// SIMATIC STEP 7 (V5.x) project Line1A_Nozzle_20101204
// CPU: CPU 315-2 DP
// station: Hardware
// station: SIMATIC 300(1)
// station: P_ADR_BUS
// station: P_ADR_BUS
// station: Configuration
// program: S7 Program(6)
// program: Controllo camera doppio
// program: Backup_prima_della_mod
// program: SIMODRIVE 611U

SYMBOL_TABLE
"Z10"	C 10	COUNTER	// Counter
"Z11"	C 11	COUNTER	// Counter
"Z12"	C 12	COUNTER	// Counter
"Z13"	C 13	COUNTER	// Counter
"DI_Balluff1"	DB 5	FB 20	// DB Instance of FB20
"DatiOP170B"	DB 7	DB 7	// PLC<->OP170B interface
"Timer"	DB 20	DB 20
"DBWork"	DB 21	DB 21
"coordinate"	DB 22	DB 22
"DB180"	DB 180	FB 24	// DB instance FB24 AsseY
"DB181"	DB 181	FB 24	// DB instance FB24 AsseX
"DBWork2"	DB 200	DB 200
"Asse_611U"	FB 16	FB 16	// Axis 611U management
"BALLUFF"	FB 20	FB 20	// BALLUFF Reader/Writer management
"FB24 - Gestione Mov Assi"	FB 24	FB 24	// GESTIONE ASSI STAZIONE
"NormalizzazioneAnalogico"	FC 7	FC 7	// Normalization of a analog value
"FC11 - STATUS"	FC 11	FC 11	// Sensors and proximity state
"FC12 - GENERAL"	FC 12	FC 12	// General management
"FC13 - MANUAL"	FC 13	FC 13	// Manual commands
"FC14 - AUTOMATIC"	FC 14	FC 14	// Automatic cycle management
"FC16 - ALARMS"	FC 16	FC 16	// Alarms management
"FC17 - OPERATOR PANNEL"	FC 17	FC 17	// Operator pannel management
"FC18 - OUTPUTS"	FC 18	FC 18	// Outputs management
"FC19 - REPOSITIONING"	FC 19	FC 19	// Repositioning management
"FC - AUTOMATIC"	FC 24	FC 24
"FC50 - TEACH-IN"	FC 50	FC 50
"FC51 - TYPE TOOL"	FC 51	FC 51
"FC52 - SYSTEM VISION"	FC 52	FC 52
"FC53 - REWORK"	FC 53	FC 53
"FC81 - GEST AXIS"	FC 81	FC 81	// Management axis
"FC117 - ERROR TOOL"	FC 117	FC 117
"TimeOut"	FC 800	FC 800	// Management TimeOut movimenti
"E0.0"	I 0.0	BOOL	// THERMAL SWTCH_ASPIRATOR_MTR
"E0.1"	I 0.1	BOOL	// 230 Vac power supply circuit braker
"E0.2"	I 0.2	BOOL	// 230 VAC PS CKT BRAKER
"E0.3"	I 0.3	BOOL	// Welding Machine OK
"E0.4"	I 0.4	BOOL	// Reserve
"E0.5"	I 0.5	BOOL	// AUXILIXARY ON
"DOOR CLOSE"	I 0.6	BOOL	// Reserve
"E0.7"	I 0.7	BOOL	// SAFETY BARRIER
"E1.0"	I 1.0	BOOL	// CYCLE_START
"E1.1"	I 1.1	BOOL	// AUTO_MANUAL
"E1.2"	I 1.2	BOOL	// COMPRESSED AIR
"E1.3"	I 1.3	BOOL	// AXIS RESET_POS
"E1.4"	I 1.4	BOOL	// Rotary table motor thermal switch
"E1.5"	I 1.5	BOOL	// LCK_UNLCK_DOORS_PB
"E1.6"	I 1.6	BOOL	// Reserve
"E1.7"	I 1.7	BOOL	// DRIVE TEMP
"E2.0"	I 2.0	BOOL	// STOP_CYCLE_PB
"E2.1"	I 2.1	BOOL	// Doors Closed & Locked
"E2.2"	I 2.2	BOOL	// Safety Barrier OK
"E2.3"	I 2.3	BOOL	// WELDING_TORCH_DWN
"E2.4"	I 2.4	BOOL	// WELDING_TORCH_UP
"E2.5"	I 2.5	BOOL	// ROTARY_TABLE_ZERO
"E2.6"	I 2.6	BOOL	// ROTARY_TABLE_ZERO1
"E2.7"	I 2.7	BOOL	// Reserve
"E3.0"	I 3.0	BOOL	// VEN DETECTOR_FWD
"E3.1"	I 3.1	BOOL	// VEN DETECTOR_REV
"E3.2"	I 3.2	BOOL	// VEN DETECTOR_DWN
"E3.3"	I 3.3	BOOL	// VEN DETECTOR_UP
"E3.4"	I 3.4	BOOL	// ROTARY_TABLE_CAM
"E3.5"	I 3.5	BOOL	// Reserve
"E3.6"	I 3.6	BOOL	// Reserve
"E3.7"	I 3.7	BOOL	// Reserve
"e5.0"	I 5.0	BOOL	// Lever Detector System - bit 0
"e5.1"	I 5.1	BOOL	// Lever Detector System - bit 1
"e5.2"	I 5.2	BOOL	// Lever Detector System - bit 2
"e5.3"	I 5.3	BOOL	// Lever Detector System - bit 3
"e5.4"	I 5.4	BOOL	// Lever Detector System - bit 4
"e5.5"	I 5.5	BOOL	// Lever Detector System - bit 5
"e5.6"	I 5.6	BOOL	// Lever Detector System - bit 6
"e5.7"	I 5.7	BOOL	// Lever Detector System - bit 7
"e6.0"	I 6.0	BOOL	// Lever Detector System - bit 8
"e6.1"	I 6.1	BOOL	// Lever Detector System - bit 9
"e6.2"	I 6.2	BOOL	// Lever Detector System - bit 10
"e6.3"	I 6.3	BOOL	// Lever Detector System - bit 11 - 12è13
"e6.4"	I 6.4	BOOL	// Lever Detector System - bit 12
"e6.5"	I 6.5	BOOL	// Lever Detector System - bit 13
"e6.6"	I 6.6	BOOL	// Lever Detector System - bit 14
"e6.7"	I 6.7	BOOL	// Lever Detector System - Vane Assy Total Number
"EXSTRACTOR_HIGH"	I 7.2	BOOL
"EXSTRACTOR_LOW"	I 7.3	BOOL
"TABLE_LCK_CYCLINDER_UP"	I 7.4	BOOL
"TABLE_LCK_CYCLINDER_DWN"	I 7.5	BOOL
"E32.0"	I 32.0	BOOL	// Push-button start cycle (on load position)
"E32.1"	I 32.1	BOOL	// Push button stop cycle
"E32.2"	I 32.2	BOOL	// Aut/Man Selector
"E32.3"	I 32.3	BOOL	// Reserve
"E32.4"	I 32.4	BOOL	// Reserve
"E32.5"	I 32.5	BOOL	// Lock/Unlock doors Push Button
"E32.6"	I 32.6	BOOL	// Reserve
"E32.7"	I 32.7	BOOL	// Air Presence
"E34.0"	I 34.0	BOOL	// Cam Table
"E34.1"	I 34.1	BOOL	// Reserve
"E34.2"	I 34.2	BOOL	// Reserve
"E34.3"	I 34.3	BOOL	// Reserve
"E34.4"	I 34.4	BOOL	// Table locker cylinder  up
"E34.5"	I 34.5	BOOL	// Table locker cylinder down
"E34.6"	I 34.6	BOOL	// Exstractor High
"E34.7"	I 34.7	BOOL	// Extractor Low
"E35.0"	I 35.0	BOOL	// Torch Welding low
"E35.1"	I 35.1	BOOL	// Torch Welding high
"E35.2"	I 35.2	BOOL	// Home Assy
"E35.3"	I 35.3	BOOL	// 1 --> PP1 on welding ; 0 --> PP2 on welding
"E35.4"	I 35.4	BOOL	// Detect components Control group High
"E35.5"	I 35.5	BOOL	// Detect components Control group Low
"E35.6"	I 35.6	BOOL	// Detect components Control group forward
"E35.7"	I 35.7	BOOL	// Detect components Control group backward
"E36.0"	I 36.0	BOOL	// Reserve not mounted
"E36.1"	I 36.1	BOOL	// Reserve not mounted
"E36.2"	I 36.2	BOOL	// Reserve not mounted
"E36.3"	I 36.3	BOOL	// Reserve not mounted
"E36.4"	I 36.4	BOOL	// Reserve not mounted
"E36.5"	I 36.5	BOOL	// Reserve not mounted
"E36.6"	I 36.6	BOOL	// Reserve not mounted
"E36.7"	I 36.7	BOOL	// Reserve not mounted
"E52.0"	I 52.0	BOOL	// Lever Detector System - bit 0
"E52.1"	I 52.1	BOOL	// Lever Detector System - bit 1
"E52.2"	I 52.2	BOOL	// Lever Detector System - bit 2
"E52.3"	I 52.3	BOOL	// Lever Detector System - bit 3
"E52.4"	I 52.4	BOOL	// Lever Detector System - bit 4
"E52.5"	I 52.5	BOOL	// Lever Detector System - bit 5
"E52.6"	I 52.6	BOOL	// Lever Detector System - bit 6
"E52.7"	I 52.7	BOOL	// Lever Detector System - bit 7
"E53.0"	I 53.0	BOOL	// Lever Detector System - bit 8
"E53.1"	I 53.1	BOOL	// Lever Detector System - bit 9
"E53.2"	I 53.2	BOOL	// Lever Detector System - bit 10
"E53.3"	I 53.3	BOOL	// Lever Detector System - bit 11 - 12è13
"E53.4"	I 53.4	BOOL	// Lever Detector System - bit 12
"E53.5"	I 53.5	BOOL	// Lever Detector System - bit 13
"E53.6"	I 53.6	BOOL	// Lever Detector System - bit 14
"E53.7"	I 53.7	BOOL	// Lever Detector System - Vane Assy Total Number
"E64.0"	I 64.0	BOOL	// VOSION SYSTEM OK
"E64.1"	I 64.1	BOOL	// Busy
"E64.2"	I 64.2	BOOL	// Or
"E64.3"	I 64.3	BOOL	// Error
"E64.4"	I 64.4	BOOL	// Gate
"E64.5"	I 64.5	BOOL	// Strobe trigger 0 out
"E64.6"	I 64.6	BOOL	// Strobe trigger 1 out
"E64.7"	I 64.7	BOOL	// DO0
"E65.0"	I 65.0	BOOL	// DO1
"E65.1"	I 65.1	BOOL	// DO2
"E65.2"	I 65.2	BOOL	// DO3
"E65.3"	I 65.3	BOOL	// DO4
"E65.4"	I 65.4	BOOL	// DO5
"E65.5"	I 65.5	BOOL	// DO6
"E65.6"	I 65.6	BOOL	// DO7
"E65.7"	I 65.7	BOOL	// DO8
"M0.0"	M 0.0	BOOL	// Clock 0,1 s
"M0.1"	M 0.1	BOOL	// Clock 0,2 s
"M0.2"	M 0.2	BOOL	// Clock 0,4 s
"M0.3"	M 0.3	BOOL	// Clock 0,5 s
"M0.4"	M 0.4	BOOL	// Clock 0,8 s
"M0.5"	M 0.5	BOOL	// Clock 1 s
"M0.6"	M 0.6	BOOL	// Clock 1,6 s
"M0.7"	M 0.7	BOOL	// Clock 2 s
"Off"	M 1.0	BOOL	// Merker always OFF
"On"	M 1.1	BOOL	// Merker always ON
"ToDo"	M 1.2	BOOL
"Bypass"	M 1.3	BOOL	// Merker that indicates a bypass forced of the code
"BypassPC"	M 1.4	BOOL	// Merker for bypass control handshake with PC supervision
"Clock_P"	M 1.5	BOOL	// Positiv pulse of clock
"Clock_N"	M 1.6	BOOL	// Negativ pulse of code
"Clock_10s"	M 1.7	BOOL	// 10 seconds clock
"M2.0"	M 2.0	BOOL	// Occhio
"BPSupervisor"	M 3.0	BOOL	// By Pass del supervisore
"Auxiliary_ON"	M 10.0	BOOL	// Auxiliary ON
"COMPRESSED_AIR"	M 10.1	BOOL	// Compressed Air
"SHIELDS_OK"	M 10.2	BOOL	// Schermi Chiusi e bloccati
"MACHINE_ON"	M 10.3	BOOL	// Machine OK
"START_POS"	M 11.0	BOOL	// Machine in initial positon
"START_POS_MEM"	M 11.1	BOOL	// mem initial position
"M11.2"	M 11.2	BOOL	// Manual Mode Selected
"SEMI"	M 11.3	BOOL	// Selezione modo semi automatico
"AUT"	M 11.4	BOOL	// Automatic Mode Selected
"START"	M 12.0	BOOL	// Start machine
"START_PULSE"	M 12.1	BOOL	// Pulse of start push-button
"SINGLE_CYCLE"	M 12.2	BOOL	// 1=ciclo singolo 0=ciclo continuo
"ALARM"	M 12.3	BOOL	// Alarm
"END_CYCLE"	M 12.4	BOOL	// Automatic cycle finished
"CmdMan_Av"	M 12.5	BOOL	// Forward manual command
"CmdMan_Ind"	M 12.6	BOOL	// Backward manual command
"STOP_BUTTON"	M 12.7	BOOL	// STATUS - stop button
"M13.0"	M 13.0	BOOL	// STATUS - Lock/Unlock doors Push Button
"M14.0"	M 14.0	BOOL	// Mem Lever Detector System - bit 0
"M14.1"	M 14.1	BOOL	// Mem Lever Detector System - bit 1
"M14.2"	M 14.2	BOOL	// Mem Lever Detector System - bit 2
"M14.3"	M 14.3	BOOL	// Mem Lever Detector System - bit 3
"M14.4"	M 14.4	BOOL	// Mem Lever Detector System - bit 4
"M14.5"	M 14.5	BOOL	// Mem Lever Detector System - bit 5
"M14.6"	M 14.6	BOOL	// Mem Lever Detector System - bit 6
"M14.7"	M 14.7	BOOL	// Mem Lever Detector System - bit 7
"M15.0"	M 15.0	BOOL	// Mem Lever Detector System - bit 8
"M15.1"	M 15.1	BOOL	// Mem Lever Detector System - bit 9
"M15.2"	M 15.2	BOOL	// Mem Lever Detector System - bit 10
"M15.3"	M 15.3	BOOL	// Mem Lever Detector System - bit 11
"M15.4"	M 15.4	BOOL	// Mem Lever Detector System - bit 12
"M15.5"	M 15.5	BOOL	// Mem Lever Detector System - bit 13
"M15.6"	M 15.6	BOOL	// Mem Lever Detector System - bit 14 (Roller)
"M15.7"	M 15.7	BOOL	// Mem Lever Detector System - bit 15
"M16.0"	M 16.0	BOOL	// mem Reworked Parts
"M16.1"	M 16.1	BOOL	// Disable Extractor if Rework
"M16.2"	M 16.2	BOOL	// Part on table 1 welding
"M16.3"	M 16.3	BOOL	// Part on Table 2 Welding
"M16.4"	M 16.4	BOOL	// Table can ROTATE
"M16.5"	M 16.5	BOOL	// Extractor can MOVE
"M16.6"	M 16.6	BOOL	// OK Extract
"M16.7"	M 16.7	BOOL	// Manual PAge Active
"M17.2"	M 17.2	BOOL	// Rework
"M17.3"	M 17.3	BOOL	// Vane no welding
"M17.4"	M 17.4	BOOL	// PP2 - OUT
"M17.5"	M 17.5	BOOL	// PP1 - OUT
"M17.6"	M 17.6	BOOL	// AUX - F R E E
"M17.7"	M 17.7	BOOL	// AUX - F R E E
"M18.0"	M 18.0	BOOL	// AUX - F R E E
"M18.1"	M 18.1	BOOL	// AUX - F R E E
"M18.2"	M 18.2	BOOL	// AUX - F R E E
"M18.3"	M 18.3	BOOL	// AUX - F R E E
"M18.4"	M 18.4	BOOL	// AUX - F R E E
"M18.5"	M 18.5	BOOL	// AUX - F R E E
"M18.6"	M 18.6	BOOL	// AUX - F R E E
"M18.7"	M 18.7	BOOL	// AUX - F R E E
"M19.0"	M 19.0	BOOL	// AUX - F R E E
"M19.1"	M 19.1	BOOL	// AUX - F R E E
"M19.2"	M 19.2	BOOL	// AUX - F R E E
"M19.3"	M 19.3	BOOL	// AUX - F R E E
"M19.4"	M 19.4	BOOL	// AUX - F R E E
"M19.5"	M 19.5	BOOL	// AUX - F R E E
"M19.6"	M 19.6	BOOL	// AUX - F R E E
"M19.7"	M 19.7	BOOL	// AUX - F R E E
"M20.0"	M 20.0	BOOL	// AUX - F R E E
"M20.1"	M 20.1	BOOL	// AUX - F R E E
"M20.2"	M 20.2	BOOL	// Presence of tool to assembly nozzle
"M20.3"	M 20.3	BOOL	// AUX - F R E E
"M20.4"	M 20.4	BOOL	// Tension OK
"M20.5"	M 20.5	BOOL	// AUX - F R E E
"M20.6"	M 20.6	BOOL	// AUX - F R E E
"M20.7"	M 20.7	BOOL	// AUX-Man
"M21.0"	M 21.0	BOOL	// STATUS - Mem Component pinched on Workrest - FC1
"Mem E34.5"	M 21.1	BOOL	// Mem Component pinched on Workrest - FC2
"M21.2"	M 21.2	BOOL	// AUX - F R E E
"M21.3"	M 21.3	BOOL	// AUX - F R E E
"M21.4"	M 21.4	BOOL	// Aux Alarm
"Warning"	M 21.5	BOOL	// Warning
"ResetAlarm"	M 21.6	BOOL	// Reset alarm
"Repos"	M 21.7	BOOL	// Repositioning
"M22.0"	M 22.0	BOOL	// STATUS - Table locker up
"M22.1"	M 22.1	BOOL	// STATUS - Table locker Down
"CmdMan_Av_Pulse"	M 22.2	BOOL	// Pulse of forward manual command
"CmdMan_Ind_Pulse"	M 22.3	BOOL	// Pulse of backward manual command
"M22.4"	M 22.4	BOOL	// Forward command
"M22.5"	M 22.5	BOOL	// Backward command
"CmdMan_Esg"	M 22.6	BOOL	// Memory of manual command executed
"CicloInCorso"	M 22.7	BOOL	// Automatic cycle in course
"M23.0"	M 23.0	BOOL	// Mem Start
"StopAEndCycle"	M 23.1	BOOL
"ChangeFunc"	M 23.2	BOOL	// Pulse change operation mode
"PresencePz"	M 23.3	BOOL
"SafetyBarrier_KO"	M 23.5	BOOL	// STATUS - Security bar KO
"M24.0"	M 24.0	BOOL	// STATUS - Torch Welding low
"M24.1"	M 24.1	BOOL	// STATUS - Torch Welding high
"M24.2"	M 24.2	BOOL	// STATUS -
"M24.3"	M 24.3	BOOL	// STATUS -
"M24.4"	M 24.4	BOOL	// STATUS - Cam table
"M24.5"	M 24.5	BOOL	// 1 --> PP1 on welding ;0 --> PP2 on welding
"M25.0"	M 25.0	BOOL	// Position Rotation 0°
"M25.1"	M 25.1	BOOL	// Position Rotation 180°
"M25.2"	M 25.2	BOOL	// Pos 0° e camma OK
"M25.3"	M 25.3	BOOL	// Pos 180° e camma OK
"M25.7"	M 25.7	BOOL	// Pulse Cam
"M26.1"	M 26.1	BOOL	// Table is FREE
"M26.2"	M 26.2	BOOL	// STATUS - System Detector Up
"M26.3"	M 26.3	BOOL	// STATUS - System Detector Lower
"M26.4"	M 26.4	BOOL	// STATUS - Detector work position
"M26.5"	M 26.5	BOOL	// STATUS - Detector park position
"M26.6"	M 26.6	BOOL	// STATUS - Exstractor High
"M26.7"	M 26.7	BOOL	// STATUS - Extractor low
"M28.0"	M 28.0	BOOL	// STATUS - DO1SYSTEM VISION
"M28.1"	M 28.1	BOOL	// STATUS - DO2 SYSTEM VISION
"M28.2"	M 28.2	BOOL	// STATUS - DO3 SYSTEM VISION
"M28.3"	M 28.3	BOOL	// STATUS - DO4 SYSTEM VISION
"M29.0"	M 29.0	BOOL	// STATUS - Run System Vision
"M29.1"	M 29.1	BOOL	// STATUS - Busy System Vision
"M29.2"	M 29.2	BOOL	// STATUS - OK System Vision
"M29.3"	M 29.3	BOOL	// STATUS - Error System Vision
"M29.4"	M 29.4	BOOL	// STATUS - Gate System Vision
"M29.6"	M 29.6	BOOL	// STATUS - DO1 SYSTEM VISION
"M29.7"	M 29.7	BOOL	// STATUS - DO0 SYSTEM VISION
"M30.0"	M 30.0	BOOL	// MAN - Table Rotation Forward
"M30.1"	M 30.1	BOOL	// MAN - Table Rotation Backward
"M30.2"	M 30.2	BOOL	// MAN - Jog + AsseY
"M30.3"	M 30.3	BOOL	// MAN - Jog - AsseY
"M30.4"	M 30.4	BOOL	// MAN - Jog + AsseX
"M30.5"	M 30.5	BOOL	// MAN - Jog - AsseX
"M30.6"	M 30.6	BOOL	// MAN - Forward SD
"M30.7"	M 30.7	BOOL	// MAN - Backward SD
"M31.0"	M 31.0	BOOL	// MAN - High SD
"M31.1"	M 31.1	BOOL	// MAN - Low SD
"M31.2"	M 31.2	BOOL	// MAN - High TW
"M31.3"	M 31.3	BOOL	// MAN - Low TW
"M31.4"	M 31.4	BOOL	// MAN - Extractor High
"M31.5"	M 31.5	BOOL	// MAN - Extractor down
"M31.6"	M 31.6	BOOL	// MAN - ON\OFF TW
"M31.7"	M 31.7	BOOL	// MAN - START/STOP WM
"M32.0"	M 32.0	BOOL	// Man  -  Start Torch W"elding
"M32.1"	M 32.1	BOOL	// MAN - Test Arco Gas Ok
"M32.2"	M 32.2	BOOL	// MAN - Test Arco Gas
"M32.3"	M 32.3	BOOL	// MAN - Torch Welding Temp Ok
"M32.4"	M 32.4	BOOL	// MAN - low table locker cylinder
"M32.5"	M 32.5	BOOL	// MAN - up table locker cylinder
"M32.6"	M 32.6	BOOL	// MAN - Welding
"M32.7"	M 32.7	BOOL	// MAN - Free
"M33.0"	M 33.0	BOOL	// MAN - Free
"M33.1"	M 33.1	BOOL	// MAN - Free
"M33.2"	M 33.2	BOOL	// MAN - Free
"M33.3"	M 33.3	BOOL	// MAN - Free
"M33.4"	M 33.4	BOOL	// MAN - Free
"M33.5"	M 33.5	BOOL	// MAN - Free
"M33.6"	M 33.6	BOOL	// MAN - Free
"M33.7"	M 33.7	BOOL	// MAN - Free
"M34.0"	M 34.0	BOOL	// MAN - Memory for rotation table
"M34.1"	M 34.1	BOOL	// MAN - Memory back rotation table
"M34.2"	M 34.2	BOOL	// MAN - Free
"M34.3"	M 34.3	BOOL	// MAN - Free
"M34.4"	M 34.4	BOOL	// MAN - Free
"M34.5"	M 34.5	BOOL	// MAN - Free
"M34.6"	M 34.6	BOOL	// MAN - Free
"M34.7"	M 34.7	BOOL	// MAN - Free
"M40.0"	M 40.0	BOOL	// RIP - Start repositioning
"M40.1"	M 40.1	BOOL	// RIP - Start reposit CamTable
"M40.2"	M 40.2	BOOL	// RIP - Cam Table
"M40.3"	M 40.3	BOOL	// RIP - System Detector vertical
"M40.4"	M 40.4	BOOL	// RIP - System Detector horizontal
"M40.5"	M 40.5	BOOL	// RIP - torch welding
"M40.6"	M 40.6	BOOL	// RIP - estractor
"M40.7"	M 40.7	BOOL	// RIP - Axis X and Y
"M41.0"	M 41.0	BOOL	// RIP - low table locker cylinder
"M41.1"	M 41.1	BOOL	// RIP - up table locker cylinder
"M41.2"	M 41.2	BOOL	// RIP - Free
"M41.3"	M 41.3	BOOL	// RIP - Free
"M41.4"	M 41.4	BOOL	// RIP - Free
"M41.5"	M 41.5	BOOL	// RIP - Free
"M41.6"	M 41.6	BOOL	// RIP - Free
"M41.7"	M 41.7	BOOL	// RIP - Free
"M42.0"	M 42.0	BOOL	// RIP - Free
"M42.1"	M 42.1	BOOL	// RIP - Table locker
"M42.2"	M 42.2	BOOL	// RIP - Free
"M42.3"	M 42.3	BOOL	// RIP - Free
"M42.4"	M 42.4	BOOL	// RIP - Free
"M42.5"	M 42.5	BOOL	// RIP - Free
"M42.6"	M 42.6	BOOL	// RIP - Free
"M42.7"	M 42.7	BOOL	// RIP - Free
"M50.0"	M 50.0	BOOL	// AUT - Table forward Side A
"M50.1"	M 50.1	BOOL	// AUT - Table backward Side B
"M50.2"	M 50.2	BOOL	// AUT - System Detector Forward
"M50.3"	M 50.3	BOOL	// AUT - System Detector Backward
"M50.4"	M 50.4	BOOL	// AUT - System Detector Low
"M50.5"	M 50.5	BOOL	// AUT - System Detector High
"M50.6"	M 50.6	BOOL	// AUT - welding down
"M50.7"	M 50.7	BOOL	// AUT - welding up
"M51.0"	M 51.0	BOOL	// AUT - Free
"M51.1"	M 51.1	BOOL	// AUT - Free
"M51.2"	M 51.2	BOOL	// AUT - Free
"M51.3"	M 51.3	BOOL	// AUT - Estractor High
"M51.4"	M 51.4	BOOL	// AUT - Estractor Low
"M51.5"	M 51.5	BOOL	// AUT - Free
"M51.6"	M 51.6	BOOL	// AUT - Free
"M51.7"	M 51.7	BOOL	// AUT - Free
"M52.0"	M 52.0	BOOL	// AUT -Temp  welding OK
"M52.1"	M 52.1	BOOL	// AUT - welding now
"M52.2"	M 52.2	BOOL	// AUT - Trigger System Vision
"M52.3"	M 52.3	BOOL	// AUT - ligth up
"M52.4"	M 52.4	BOOL	// AUT - Test Arc
"M52.5"	M 52.5	BOOL	// AUT - Test Arc Gas Ok
"M52.6"	M 52.6	BOOL	// AUT - low table locker cylinder
"M52.7"	M 52.7	BOOL	// AUT - up table locker cylinder
"M53.0"	M 53.0	BOOL	// AUT - Table locker Up
"M53.1"	M 53.1	BOOL	// AUT - Table locker Down
"M60.0"	M 60.0	BOOL	// STEP - 1:Table Forward
"M60.1"	M 60.1	BOOL	// STEP - 2:System Detector Forward
"M60.2"	M 60.2	BOOL	// STEP 3- System Detector Low
"M60.3"	M 60.3	BOOL	// STEP - 3 Check Nozzle Component
"M60.4"	M 60.4	BOOL	// STEP - 5 System detector High
"M60.5"	M 60.5	BOOL	// STEP 6 - System Detector Bacward
"M60.6"	M 60.6	BOOL	// STEP -7 welding down on point
"M60.7"	M 60.7	BOOL	// STEP - welding OK
"M61.0"	M 61.0	BOOL	// STEP - All welding is effectuated
"M61.1"	M 61.1	BOOL	// STEP - Photo Executed
"M61.2"	M 61.2	BOOL	// STEP - Axis in position 0
"M61.3"	M 61.3	BOOL	// STEP - point for welding receive
"M61.4"	M 61.4	BOOL	// STEP - welding up after work
"M61.5"	M 61.5	BOOL	// STEP - Welding in progress
"M61.6"	M 61.6	BOOL	// STEP - Start Rotation Table
"M61.7"	M 61.7	BOOL	// STEP - Photo without error
"M62.0"	M 62.0	BOOL	// STEP - Mem Reset Table
"M62.1"	M 62.1	BOOL	// STEP - Free
"M62.2"	M 62.2	BOOL	// STEP - Table cylinder up
"M62.3"	M 62.3	BOOL	// STEP - Free
"M62.4"	M 62.4	BOOL	// STEP - Free
"M62.5"	M 62.5	BOOL	// STEP - Free
"M62.6"	M 62.6	BOOL	// STEP - Free
"M62.7"	M 62.7	BOOL	// STEP - Photo Executed
"M63.0"	M 63.0	BOOL	// STEP - Nozzle Extracted
"M63.1"	M 63.1	BOOL	// STEP - Table Cylinder Low
"M63.6"	M 63.6	BOOL	// STEP - receive point photo
"M66.0"	M 66.0	BOOL	// STEP - photo 1 is NO good
"M66.1"	M 66.1	BOOL	// STEP - photo 2 is NO good
"M66.4"	M 66.4	BOOL	// STEP - Axis in position
"M66.6"	M 66.6	BOOL	// STEP - Execute 2th photo
"M66.7"	M 66.7	BOOL	// STEP - All photo is NO Good
"M67.0"	M 67.0	BOOL	// STEP - Axis Y in position
"M67.1"	M 67.1	BOOL	// STEP - Axis X in position
"M70.0"	M 70.0	BOOL	// Nozzle components Ok
"M70.1"	M 70.1	BOOL	// memNozzle-components Ok
"M70.2"	M 70.2	BOOL	// Component of Nozzle KO
"M70.3"	M 70.3	BOOL	// error assembling su PP1
"M70.4"	M 70.4	BOOL	// error assembling su PP2
"M71.0"	M 71.0	BOOL	// System Detector in Pos initial
"M72.0"	M 72.0	BOOL	// ready for welding
"M73.0"	M 73.0	BOOL	// Enable velocity for repositioning
"M74.0"	M 74.0	BOOL	// Output SV enable
"M74.1"	M 74.1	BOOL	// piece good
"M74.2"	M 74.2	BOOL	// piece reject
"M75.0"	M 75.0	BOOL	// Enable movement axis for teach in
"M75.1"	M 75.1	BOOL	// TeachIn OK
"M76.0"	M 76.0	BOOL	// position welding receive
"MEM Welding Machine OK"	M 80.0	BOOL
"Type_PP1_10_vane"	M 90.0	BOOL	// PP1-10 presence
"Type_PP2_9_vane"	M 90.1	BOOL	// presence PP2 -11 welding
"Type_PP3_9_vane"	M 90.2	BOOL	// presence PP3 - 9welding
"Type_PP4_13_vane"	M 90.3	BOOL	// presence PP4 - 13 Welding
"AUT STEP 1"	M 160.0	BOOL
"AUT STEP 2"	M 160.1	BOOL
"AUT STEP 3"	M 160.2	BOOL
"AUT STEP 4"	M 160.3	BOOL
"AUT STEP 5"	M 160.4	BOOL
"AUT STEP 6"	M 160.5	BOOL
"AUT STEP 7"	M 160.6	BOOL
"AUT STEP 8"	M 160.7	BOOL
"AUT STEP 9"	M 161.0	BOOL
"AUT STEP10"	M 161.1	BOOL
"AUT STEP11"	M 161.2	BOOL
"AUT STEP12"	M 161.3	BOOL
"AUT STEP13"	M 161.4	BOOL
"AUT STEP14"	M 161.5	BOOL
"AUT STEP15"	M 161.6	BOOL
"AUT STEP16"	M 161.7	BOOL
"AUT STEP17"	M 162.0	BOOL
"AUT STEP18"	M 162.1	BOOL
"AUT STEP19"	M 162.2	BOOL
"AUT STEP20"	M 162.3	BOOL
"AUT STEP21"	M 162.4	BOOL
"AUT STEP22"	M 162.5	BOOL
"AUT STEP23"	M 162.6	BOOL
"AUT STEP24"	M 162.7	BOOL
"AUT STEP25"	M 163.0	BOOL
"AUT STEP26"	M 163.1	BOOL
"AUT STEP27"	M 163.2	BOOL
"AUT STEP28"	M 163.3	BOOL
"AUT STEP29"	M 163.4	BOOL
"AUT STEP30"	M 163.5	BOOL
"Clock 0.5 S"	M 200.3	BOOL
"Clock 1s"	M 200.5	BOOL
"M254.0"	M 254.0	BOOL	// Front Command HOME
"M254.1"	M 254.1	BOOL	// Front Command END
"M256.0"	M 256.0	BOOL	// Pulse
"M256.2"	M 256.2	BOOL	// Pulse
"M256.6"	M 256.6	BOOL	// Pulse
"M256.7"	M 256.7	BOOL	// Pulse
"M340.0"	M 340.0	BOOL	// AXIS Y:STOP MOVE
"M340.1"	M 340.1	BOOL	// AXIS Y:START POSITIONING
"M340.2"	M 340.2	BOOL	// AXIS Y:START SEARCH HOME
"M340.3"	M 340.3	BOOL	// AXIS Y:START POSITIONING ON HOME
"M340.4"	M 340.4	BOOL	// AXIS X:COMMAND JOG PLUS
"M340.5"	M 340.5	BOOL	// AXIS X:COMANDO JOG LESS
"M341.0"	M 341.0	BOOL	// AXIS Y:ACHIEVED LOCATION
"M341.1"	M 341.1	BOOL	// AXIS Y:REFERED AXIS
"M341.2"	M 341.2	BOOL	// AXIS Y:AXIS LOCATION ON HOME
"M341.3"	M 341.3	BOOL	// AXIS Y:AXIS STOP NONE COMMAND PROGRESS
"M341.4"	M 341.4	BOOL	// AXIS Y:SETTING SETTING IN MOTION OK
"M341.5"	M 341.5	BOOL	// AXIS Y:ALLRM SETTING IN MOTION
"M342.0"	M 342.0	BOOL	// AXIS Y:AXIS ON CAM OF  REFERENCE
"M342.1"	M 342.1	BOOL	// AXIS Y:AXIS ON OVER RACE NEGATIVE HARDWARE
"M342.2"	M 342.2	BOOL	// AXIS Y:AXIS ON OVER RACE POSITIVE HARDWARE
"M342.3"	M 342.3	BOOL	// AXIS Y:COMMAND BRAKE PARKING
"M342.4"	M 342.4	BOOL	// AXIS Y:AXIS ON OVER RACE NEGATIVE SOFTWARE
"M342.5"	M 342.5	BOOL	// AXIS Y:AXIS ON OVER RACE POSITIVE SOFTWARE
"M342.6"	M 342.6	BOOL	// AXIS Y:POSSIBLE MOVE AXIS
"M342.7"	M 342.7	BOOL	// AXIS Y:INITIAL LOCATION AXIS
"M343.0"	M 343.0	BOOL	// AXIS Y:START POSITIONING INCREMENTAL
"M346.0"	M 346.0	BOOL	// AXIS X:STOP MOVE
"M346.1"	M 346.1	BOOL	// AXIS X:START POSITIONING
"M346.2"	M 346.2	BOOL	// AXIS X:START SEARCH HOME
"M346.3"	M 346.3	BOOL	// AXIS X:START POSITIONING ON HOME
"M346.4"	M 346.4	BOOL	// AXIS Y:COMMAND JOG PLUS
"M346.5"	M 346.5	BOOL	// AXIS Y:COMANDO JOG LESS
"M347.0"	M 347.0	BOOL	// AXIS X:ACHIEVED LOCATION
"M347.1"	M 347.1	BOOL	// AXIS X:REFERED AXIS
"M347.2"	M 347.2	BOOL	// AXIS X:AXIS LOCATION ON HOME
"M347.3"	M 347.3	BOOL	// AXIS X:AXIS STOP NONE COMMAND PROGRESS
"M347.4"	M 347.4	BOOL	// AXIS X:SETTING SETTING IN MOTION OK
"M347.5"	M 347.5	BOOL	// AXIS X:ALLRM SETTING IN MOTION
"M348.0"	M 348.0	BOOL	// AXIS X:AXIS ON CAM OF  REFERENCE
"M348.1"	M 348.1	BOOL	// AXIS X:AXIS ON OVER RACE NEGATIVE HARDWARE
"M348.2"	M 348.2	BOOL	// AXIS X:AXIS ON OVER RACE POSITIVE HARDWARE
"M348.3"	M 348.3	BOOL	// AXIS X:COMMAND BRAKE PARKING
"M348.4"	M 348.4	BOOL	// AXIS X:AXIS ON OVER RACE NEGATIVE SOFTWARE
"M348.5"	M 348.5	BOOL	// AXIS X:AXIS ON OVER RACE POSITIVE SOFTWARE
"M348.6"	M 348.6	BOOL	// AXIS X:POSSIBLE MOVE AXIS
"M348.7"	M 348.7	BOOL	// AXIS X:INITIAL LOCATION AXIS
"M349.0"	M 349.0	BOOL	// AXIS X:START POSITIONING INCREMENTAL
"Photo 2 executed"	M 500.0	BOOL	// m61.1
"TriggerVisSystem2"	M 500.1	BOOL
"ErroreCamera"	M 500.7	BOOL
"M1000.0"	M 1000.0	BOOL	// AUX
"M1000.1"	M 1000.1	BOOL	// AUX
"M1000.2"	M 1000.2	BOOL	// AUX
"M1000.3"	M 1000.3	BOOL	// AUX
"M1000.4"	M 1000.4	BOOL	// AUX
"M1000.5"	M 1000.5	BOOL	// AUX
"M1000.6"	M 1000.6	BOOL	// AUX
"M1000.7"	M 1000.7	BOOL	// AUX
"M1001.0"	M 1001.0	BOOL	// AUX
"M1001.1"	M 1001.1	BOOL	// AUX
"M1001.2"	M 1001.2	BOOL	// AUX
"M1001.3"	M 1001.3	BOOL	// AUX
"M1001.4"	M 1001.4	BOOL	// AUX
"M1001.5"	M 1001.5	BOOL	// AUX
"M1001.6"	M 1001.6	BOOL	// AUX
"M1001.7"	M 1001.7	BOOL	// AUX
"M1002.0"	M 1002.0	BOOL	// AUX
"M1002.1"	M 1002.1	BOOL	// AUX
"M1002.2"	M 1002.2	BOOL	// AUX
"M1002.3"	M 1002.3	BOOL	// AUX
"M1002.4"	M 1002.4	BOOL	// AUX
"M1002.5"	M 1002.5	BOOL	// AUX
"M1002.6"	M 1002.6	BOOL	// AUX
"M1002.7"	M 1002.7	BOOL	// AUX
"M1003.0"	M 1003.0	BOOL	// AUX
"M1003.1"	M 1003.1	BOOL	// AUX
"M1003.2"	M 1003.2	BOOL	// AUX
"M1003.3"	M 1003.3	BOOL	// AUX
"M1003.4"	M 1003.4	BOOL	// AUX
"M1003.5"	M 1003.5	BOOL	// AUX
"M1003.6"	M 1003.6	BOOL	// AUX
"M1003.7"	M 1003.7	BOOL	// AUX
"M1004.0"	M 1004.0	BOOL	// AUX
"M1004.1"	M 1004.1	BOOL	// AUX
"M1004.2"	M 1004.2	BOOL	// AUX
"M1004.3"	M 1004.3	BOOL	// AUX
"M1004.4"	M 1004.4	BOOL	// AUX
"M1004.5"	M 1004.5	BOOL	// AUX
"M1004.6"	M 1004.6	BOOL	// AUX
"M1004.7"	M 1004.7	BOOL	// AUX
"M1005.0"	M 1005.0	BOOL	// AUX
"M1005.1"	M 1005.1	BOOL	// AUX
"M1005.2"	M 1005.2	BOOL	// AUX
"M1005.3"	M 1005.3	BOOL	// AUX
"M1005.4"	M 1005.4	BOOL	// AUX
"M1005.5"	M 1005.5	BOOL	// AUX
"M1005.6"	M 1005.6	BOOL	// AUX
"M1005.7"	M 1005.7	BOOL	// AUX
"M1006.0"	M 1006.0	BOOL	// AUX
"M1006.1"	M 1006.1	BOOL	// AUX
"M1006.2"	M 1006.2	BOOL	// AUX
"M1006.3"	M 1006.3	BOOL	// AUX
"M1006.4"	M 1006.4	BOOL	// AUX
"M1006.5"	M 1006.5	BOOL	// AUX
"M1006.6"	M 1006.6	BOOL	// AUX
"M1006.7"	M 1006.7	BOOL	// AUX
"M1007.0"	M 1007.0	BOOL	// AUX
"M1007.1"	M 1007.1	BOOL	// AUX
"M1007.2"	M 1007.2	BOOL	// AUX
"M1007.3"	M 1007.3	BOOL	// AUX
"M1007.4"	M 1007.4	BOOL	// AUX
"M1007.5"	M 1007.5	BOOL	// AUX
"M1007.6"	M 1007.6	BOOL	// AUX
"M1007.7"	M 1007.7	BOOL	// AUX
"M1008.0"	M 1008.0	BOOL	// AUX
"M1008.1"	M 1008.1	BOOL	// AUX
"M1008.2"	M 1008.2	BOOL	// AUX
"M1008.3"	M 1008.3	BOOL	// AUX
"M1008.4"	M 1008.4	BOOL	// AUX
"M1008.5"	M 1008.5	BOOL	// AUX
"M1008.6"	M 1008.6	BOOL	// AUX
"M1008.7"	M 1008.7	BOOL	// AUX
"M1009.0"	M 1009.0	BOOL	// AUX
"M1009.1"	M 1009.1	BOOL	// AUX
"M1009.2"	M 1009.2	BOOL	// AUX
"M1009.3"	M 1009.3	BOOL	// AUX
"M1009.4"	M 1009.4	BOOL	// AUX
"M1009.5"	M 1009.5	BOOL	// AUX
"M1009.6"	M 1009.6	BOOL	// AUX
"M1009.7"	M 1009.7	BOOL	// AUX
"FPAuxON_force_Axis_reset"	M 1900.0	BOOL
"Luce telecamera"	M 1900.2	BOOL
"AppoFP_M1900.3"	M 1900.3	BOOL
"Soffio Camera"	M 1900.4	BOOL
"Manual_cameralight_on"	M 1900.5	BOOL
"M2034.0"	M 2034.0	BOOL	// Key Start from pannell
"M2034.1"	M 2034.1	BOOL	// Key Finish from pannell
"M2034.2"	M 2034.2	BOOL	// Key Teach In from Pannell
"M2034.5"	M 2034.5	BOOL	// Key Enter teach from pannel
"M2034.6"	M 2034.6	BOOL	// Key Exit teach from pannel
"M2034.7"	M 2034.7	BOOL	// Key Rite from pannell
"M2035.0"	M 2035.0	BOOL	// Key Start from Teach In page
"M2035.1"	M 2035.1	BOOL	// Key Welding Run from pannel
"M2035.2"	M 2035.2	BOOL	// Key ACK on page 21 from pannell
"MB2046"	MB 2046	BYTE	// white byte
"MD30"	MD 30	DWORD	// DWORD Manual Commands
"MD100"	MD 100	DWORD	// temp
"MD588"	MD 588	DINT	// temporary for X point
"MD592"	MD 592	DINT	// temporary for X point
"MD596"	MD 596	DINT	// target X
"MD600"	MD 600	DINT	// target Y
"MD620"	MD 620	DWORD	// InsertPointX
"MD624"	MD 624	DWORD	// InsertPointY
"MD650"	MD 650	DINT	// axis X actual position
"MD654"	MD 654	DINT	// axis Y actual posiion
"SaldEffet"	MW 110	WORD	// number welding make
"MW120"	MW 120	INT	// number welding make
"MW300"	MW 300	INT	// number point to want go
"MW2042"	MW 2042	INT	// temp for clock
"MAIN PROGRAM"	OB 1	OB 1	// Main Program
"I/O_FLT1"	OB 82	OB 82	// I/O Point Fault 1
"RACK_FLT"	OB 86	OB 86	// Loss of Rack Fault
"COMPLETE RESTART"	OB 100	OB 100	// Complete Restart
"MOD_ERR"	OB 122	OB 122	// Module Access Error
"A0.0"	Q 0.0	BOOL	// Red Lamp
"A0.1"	Q 0.1	BOOL	// Yellow Lamp
"A0.2"	Q 0.2	BOOL	// Green Lamp
"A0.3"	Q 0.3	BOOL	// Lock doors relay
"A0.4"	Q 0.4	BOOL	// Simodrive Reset realy
"A0.5"	Q 0.5	BOOL	// Reserve
"A0.6"	Q 0.6	BOOL	// Reserve
"A0.7"	Q 0.7	BOOL	// Reserve
"A1.0"	Q 1.0	BOOL	// Enable Coral Vacuum
"A1.1"	Q 1.1	BOOL	// Test Gas Arco Pilota
"A1.2"	Q 1.2	BOOL	// Forward table rotation
"A1.3"	Q 1.3	BOOL	// Backward table rotation
"A1.4"	Q 1.4	BOOL	// Enable Axis X
"A1.5"	Q 1.5	BOOL	// Enable Axis Y
"A1.6"	Q 1.6	BOOL	// Start Welding
"A1.7"	Q 1.7	BOOL	// Ignition torch
"A2.0"	Q 2.0	BOOL	// Reserve
"A2.1"	Q 2.1	BOOL	// Reserve
"A2.2"	Q 2.2	BOOL	// Reserve
"A2.3"	Q 2.3	BOOL	// Reserve
"A2.4"	Q 2.4	BOOL	// Reserve
"A2.5"	Q 2.5	BOOL	// Reserve
"A2.6"	Q 2.6	BOOL	// Reserve
"A2.7"	Q 2.7	BOOL	// Reserve
"A3.0"	Q 3.0	BOOL	// Reserve
"A3.1"	Q 3.1	BOOL	// Reserve
"A3.2"	Q 3.2	BOOL	// Reserve
"A3.3"	Q 3.3	BOOL	// Reserve
"A3.4"	Q 3.4	BOOL	// Reserve
"A3.5"	Q 3.5	BOOL	// Reserve
"A3.6"	Q 3.6	BOOL	// Reserve
"A3.7"	Q 3.7	BOOL	// Reserve
"SIMODRIVE_RESET"	Q 12.0	BOOL
"BUZZER"	Q 12.1	BOOL
"Torch Welding Machin"	Q 12.2	BOOL	// Down
"Torch Welding MachinE"	Q 12.3	BOOL	// UP
"TABLE_LCKER_DWN"	Q 12.4	BOOL
"Table locker cylinder up"	Q 12.5	BOOL
"FWD_LEVER_DETECT_SYS"	Q 12.6	BOOL
"REV_LEVER_DETECT_SYS"	Q 12.7	BOOL
"UP_lever detector system"	Q 13.0	BOOL
"DW_lever detector sys"	Q 13.1	BOOL
"UP_Down _Extractor"	Q 13.2	BOOL
"_soffio_telecamera"	Q 13.3	BOOL
"DRIVE_ENABLE"	Q 13.5	BOOL
"ENABLE_Y_AXIS"	Q 13.6	BOOL
"ENABLE_X_AXIS"	Q 13.7	BOOL
"STOP_CYCLE_LAMP"	Q 14.3	BOOL
"START_CYCLE_LAMP"	Q 14.4	BOOL
"a14.5"	Q 14.5	BOOL
"ACCESES_BARRIER_LAMP"	Q 14.6	BOOL
"Enable Coral Vacuum"	Q 17.0	BOOL
"FWD_TABLE_ROTATION"	Q 17.1	BOOL
"REVERSE_TABLE_ROTATION"	Q 17.2	BOOL
"IGNITION_TORCH"	Q 17.5	BOOL
"START_WELDING"	Q 17.6	BOOL
"Test Gas Arc Pilota"	Q 17.7	BOOL
"PLC READY"	Q 18.0	BOOL	// ADDITION
"_Illumin_telecamera"	Q 18.1	BOOL
"PIECE_REFUSE"	Q 18.3	BOOL
"RED_LAMP"	Q 18.4	BOOL
"PIECE_GOOD"	Q 18.5	BOOL
"Lamp_Door_Locked"	Q 18.6	BOOL
"LOCK_DOORS_RELAY"	Q 18.7	BOOL
"A32.0"	Q 32.0	BOOL	// Lamp Start cycle
"A32.1"	Q 32.1	BOOL	// Lamp Stop cycle
"A32.2"	Q 32.2	BOOL	// Piece Good
"A32.3"	Q 32.3	BOOL	// Piece Refuse
"A32.4"	Q 32.4	BOOL	// Unlocked doors
"A32.5"	Q 32.5	BOOL	// Emergency Lamp
"A32.6"	Q 32.6	BOOL	// Access barrier Lamp
"A32.7"	Q 32.7	BOOL	// Buzzer
"A33.0"	Q 33.0	BOOL	// Reserve
"A33.1"	Q 33.1	BOOL	// Reserve
"A33.2"	Q 33.2	BOOL	// Reserve
"A33.3"	Q 33.3	BOOL	// Reserve
"A33.4"	Q 33.4	BOOL	// Reserve not mounted
"A33.5"	Q 33.5	BOOL	// Reserve not mounted
"A33.6"	Q 33.6	BOOL	// Reserve not mounted
"A33.7"	Q 33.7	BOOL	// Reserve not mounted
"A34.0"	Q 34.0	BOOL	// Forward lever detector System
"A34.1"	Q 34.1	BOOL	// Backward lever detector System
"A34.2"	Q 34.2	BOOL	// Down lever detector system
"A34.3"	Q 34.3	BOOL	// Up lever detector system
"A34.4"	Q 34.4	BOOL	// Down Torch Welding Machine
"A34.5"	Q 34.5	BOOL	// Up Torch Welding Machine
"A34.6"	Q 34.6	BOOL	// Down Extractor
"A34.7"	Q 34.7	BOOL	// Up Extractor
"A35.0"	Q 35.0	BOOL	// Table locker down
"A35.1"	Q 35.1	BOOL	// Table locker up
"A35.2"	Q 35.2	BOOL	// Reserve
"A35.3"	Q 35.3	BOOL	// Reserve
"A35.4"	Q 35.4	BOOL	// Reserve
"A35.5"	Q 35.5	BOOL	// Reserve
"A35.6"	Q 35.6	BOOL	// Reserve
"A35.7"	Q 35.7	BOOL	// Reserve
"A64.0"	Q 64.0	BOOL	// Reset
"A64.1"	Q 64.1	BOOL	// Trigger
"A64.2"	Q 64.2	BOOL	// Data Send Request
"A64.3"	Q 64.3	BOOL	// DI0
"A64.4"	Q 64.4	BOOL	// DI1
"A64.5"	Q 64.5	BOOL	// DI2
"A64.6"	Q 64.6	BOOL	// DI3
"A64.7"	Q 64.7	BOOL	// DI4
"A65.0"	Q 65.0	BOOL	// DI5
"A65.1"	Q 65.1	BOOL	// DI6
"A65.2"	Q 65.2	BOOL	// DI7
"A65.3"	Q 65.3	BOOL	// DI8
"A65.4"	Q 65.4	BOOL	// DI9
"A65.5"	Q 65.5	BOOL	// Reserve
"A65.6"	Q 65.6	BOOL	// Reserve
"A65.7"	Q 65.7	BOOL	// Reserve
"TON"	SFB 4	SFB 4	// Generate an On Delay
"READ_CLK"	SFC 1	SFC 1	// Read System Clock
"DPRD_DAT"	SFC 14	SFC 14	// Read Consistent Data of a Standard DP Slave
"DPWR_DAT"	SFC 15	SFC 15	// Write Consistent Data to a Standard DP Slave
"BLKMOV"	SFC 20	SFC 20	// Copy Variables
"FILL"	SFC 21	SFC 21	// Initialize a Memory Area
"CREAT_DB"	SFC 22	SFC 22	// Create Data Block
"DIS_AIRT"	SFC 41	SFC 41	// Delay the Higher Priority Interrupts and Asynchronous Errors
"EN_AIRT"	SFC 42	SFC 42	// Enable Higher Priority Interrupts and Asynchronous Errors
"STP"	SFC 46	SFC 46	// Change the CPU to STOP
"LGC_GADR"	SFC 49	SFC 49	// Query the Module Slot Belonging to a Logical Address
"RDSYSST"	SFC 51	SFC 51	// Read a System Status List or Partial List
"WR_REC"	SFC 58	SFC 58	// Write Data Record
"RD_REC"	SFC 59	SFC 59	// Read a Data Record
"T2"	T 2	TIMER
"T3"	T 3	TIMER	// Time for Component Start UP
"T10"	T 10	TIMER	// Delay
"T11"	T 11	TIMER
"T12"	T 12	TIMER	// delay next step
"T13"	T 13	TIMER	// Delay
"T14"	T 14	TIMER	// timer for delay KO
"T15"	T 15	TIMER	// Delay
"T16"	T 16	TIMER	// Delay
"T17"	T 17	TIMER	// timer delay
"T18"	T 18	TIMER	// Delay
"T19"	T 19	TIMER	// delay
"T20"	T 20	TIMER	// timer delay
"T21"	T 21	TIMER	// Time Test Arc
"T22"	T 22	TIMER	// Delay
"T23"	T 23	TIMER	// Timer for repositioning
"T24"	T 24	TIMER	// Delay make 2th photo
"T25"	T 25	TIMER	// delay
"T26"	T 26	TIMER	// time for reset output rotation table
"T27"	T 27	TIMER	// Timer for Executed Photo
"T28"	T 28	TIMER	// Delay for entry in teach in mode
"T29"	T 29	TIMER	// delay for reset both axis
"T30"	T 30	TIMER	// timer dealy
"T31"	T 31	TIMER	// MAN - time for welding
"T32"	T 32	TIMER	// MAN - time for welding UP
"T33"	T 33	TIMER	// Delay
"T34"	T 34	TIMER	// Time Test Arco
"T35"	T 35	TIMER	// Delay
"T36"	T 36	TIMER	// delay for cam not present
"T37"	T 37	TIMER	// Time Torch Welding Ok
"T38"	T 38	TIMER	// timer reset alarms axis X
"T39"	T 39	TIMER	// timer reset alarms axis Y
"T40"	T 40	TIMER	// Time Torch Welding Ok
"T41"	T 41	TIMER	// delay alarm air pressure
"T42"	T 42	TIMER	// Timer stop welding
"T43"	T 43	TIMER	// Timer welding Manual
"T44"	T 44	TIMER	// Delay
"T45"	T 45	TIMER	// timer for upgrade value
"T46"	T 46	TIMER	// delay enable axis Ytimer reset alarms axis X
"T47"	T 47	TIMER	// delay
"T48"	T 48	TIMER	// delay enable axis Ytimer reset alarms axis Y
"T50"	T 50	TIMER	// Delay
"T51"	T 51	TIMER
"T52"	T 52	TIMER	// wait after rotation table
"T53"	T 53	TIMER	// delay for chek camera point
"T54"	T 54	TIMER	// delay turn OFF Buzzer
"T60"	T 60	TIMER	// Delay for entry in teach in mode
"T61"	T 61	TIMER	// delay go in position for 2th photo
"T62"	T 62	TIMER	// delay for axis in position
"T63"	T 63	TIMER	// Delay
"T_SystemDetectorDW"	T 70	TIMER
"T_SystemDetector_UP"	T 71	TIMER
"T90"	T 90	TIMER	// delay allarm for Simodrive
"VAT_1"	VAT 1	
"Coordinate_saldatura"	VAT 2	
"I/O System Vision"	VAT 3	
"Saldatrice"	VAT 4	
"VAT_12"	VAT 5	
"VAT_PUNTI_AVV"	VAT 6	
"VAT_PUNTI_AVV_2"	VAT 7	
"DB22_SaldaturaSilv"	VAT 8	
"DB22_Sald_PP1"	VAT 9	
"VAT_tool check"	VAT 10	
"VAT_Balluff"	VAT 11	
"ASSE_P"	VAT 12	
"DB22_Sald_PP3"	VAT 13	
"VAT_Point"	VAT 14	
"VAT_Point 16"	VAT 15	
"DB22_Sald_PP16"	VAT 16	
"VAT_17"	VAT 17	
"Tipo portapezzo"	VAT 18	
"VAT_Daniele"	VAT 19	
END_SYMBOL_TABLE

FUNCTION_BLOCK "Asse_611U"	// FB 16
TITLE = Axis 611U management
VERSION : 0.1
VAR_INPUT
  IO_LAddr : INT ;	//Logic address of the inputs/outputs
END_VAR
VAR
  In_Profibus : STRUCT 	//Inputs from 611U (via Profibus)
   PKW : STRUCT 	//Parameter area of the Profibus telegram
    PKE : WORD ;
    IND : WORD ;
    PWE : DINT ;
   END_STRUCT ;
   PZD : STRUCT 	//Process data area of the Profibus telegram
    ZSW1 : STRUCT 	//Status word 1
     Bit8 : BOOL ;	//Following error (0=following error outside the window error)
     Bit9 : BOOL ;	//DP control requested (1=DP master is requested to accept control)
     Bit10 : BOOL ;	//Reference position reached (1=end of traversing block reached)
     Bit11 : BOOL ;	//Reference point set (1=axis is referenced)
     Bit12 : BOOL ;	//Setpoint acknowledge (1=the traversing task is processed)
     Bit13 : BOOL ;	//Drive stationery (1=drive is not in movement)
     Bit14 : BOOL ;	//External block change selected
     Bit15 : BOOL ;	//Request passive referencing
     Bit0 : BOOL ;	//Ready to switch-on (1=ready to power-up)
     Bit1 : BOOL ;	//Ready or no fault (1=drive ready or no fault present)
     Bit2 : BOOL ;	//Controller enable (1=speed controller active and setpoint can be accepted)
     Bit3 : BOOL ;	//Fault present (1=fault present)
     Bit4 : BOOL ;	//No OFF2 (1=OFF2 not present)
     Bit5 : BOOL ;	//No OFF3 (1=OFF3 not present)
     Bit6 : BOOL ;	//Switch-on inhibit (1=power-on inhibit)
     Bit7 : BOOL ;	//Alarm present (1=alarm present)
    END_STRUCT ;
    AktSatz : STRUCT 	//Actual block status word
     Bit8 : BOOL ;	//Reserved
     Bit9 : BOOL ;	//Reserved
     Bit10 : BOOL ;	//Reserved
     Bit11 : BOOL ;	//Reserved
     Bit12 : BOOL ;	//Reserved
     Bit13 : BOOL ;	//Reserved
     Bit14 : BOOL ;	//Reserved
     Bit15 : BOOL ;	//MDI Active
     Bit0 : BOOL ;	//Bit 0 block selected
     Bit1 : BOOL ;	//Bit 1 block selected
     Bit2 : BOOL ;	//Bit 2 block selected
     Bit3 : BOOL ;	//Bit 3 block selected
     Bit4 : BOOL ;	//Bit 4 block selected
     Bit5 : BOOL ;	//Bit 5 block selected
     Bit6 : BOOL ;	//Reserved
     Bit7 : BOOL ;	//Reserved
    END_STRUCT ;
    PosZsw : STRUCT 	//Position status word
     Bit8 : BOOL ;	//Cam switching signal 1
     Bit9 : BOOL ;	//Cam switching signal 2
     Bit10 : BOOL ;	//Direct output 1 via the traversing block
     Bit11 : BOOL ;	//Direct output 2 via the traversing block
     Bit12 : BOOL ;	//Fixed endstop reached
     Bit13 : BOOL ;	//Fixed endstop clamping torque reached
     Bit14 : BOOL ;	//Traverse to fixed endstop active
     Bit15 : BOOL ;	//Teach-In executed
     Bit0 : BOOL ;	//Tracking mode active (1=tracking mode active)
     Bit1 : BOOL ;	//Velocity limiting (1=velocity is limited)
     Bit2 : BOOL ;	//Setpoint stationary (1=axis stationary on the setpoint side)
     Bit3 : BOOL ;	//In synchronism (1=slave drive is synchronized with the master drive)
     Bit4 : BOOL ;	//Axis moves forwards
     Bit5 : BOOL ;	//Axis moves backwards
     Bit6 : BOOL ;	//Minus software limit switch actuated
     Bit7 : BOOL ;	//Plus software limit switch actuated
    END_STRUCT ;
    ZSW2 : STRUCT 	//Status word 2
     Bit8 : BOOL ;	//Suppress fault 608 active
     Bit9 : BOOL ;	//n.u. (used only in the n-set mode)
     Bit10 : BOOL ;	//n.u. (used only in the n-set mode)
     Bit11 : BOOL ;	//n.u. (used only in the n-set mode)
     Bit12 : BOOL ;	//Slave sign-of-life
     Bit13 : BOOL ;	//Slave sign-of-life
     Bit14 : BOOL ;	//Slave sign-of-life
     Bit15 : BOOL ;	//Slave sign-of-life
     Bit0 : BOOL ;	//Bit 0 parameter set
     Bit1 : BOOL ;	//Bit 1 parameter set
     Bit2 : BOOL ;	//Bit 2 parameter set
     Bit3 : BOOL ;	//First speed setpoint filter inactive
     Bit4 : BOOL ;	//Rump-function generator inactive
     Bit5 : BOOL ;	//Open holding brake
     Bit6 : BOOL ;	//Integrator inhibit
     Bit7 : BOOL ;	//Parking axis selected
    END_STRUCT ;
    XretrP : DINT ;	//Actual position value
    DIG_IN : STRUCT 	//Digital inputs status
     Bit8 : BOOL ;
     Bit9 : BOOL ;
     Bit10 : BOOL ;
     Bit11 : BOOL ;
     Bit12 : BOOL ;
     Bit13 : BOOL ;
     Bit14 : BOOL ;
     Bit15 : BOOL ;
     Bit0 : BOOL ;	//Axis on home cam
     Bit1 : BOOL ;	//Axis on minus extra-corse limit switch
     Bit2 : BOOL ;	//Axis on plus extra-corse limit switch
     Bit3 : BOOL ;
     Bit4 : BOOL ;
     Bit5 : BOOL ;
     Bit6 : BOOL ;
     Bit7 : BOOL ;
    END_STRUCT ;
   END_STRUCT ;
  END_STRUCT ;
  Out_Profibus : STRUCT 	//Outputs to 611U (via Profibus)
   PKW : STRUCT 	//Parameter area of the Profibus telegram
    PKE : WORD ;
    IND : WORD ;
    PWE : DINT ;
   END_STRUCT ;
   PZD : STRUCT 	//Process data area of the Profibus telegram
    STW1 : STRUCT 	//Control word 1
     Bit8 : BOOL ;	//JOG1 (1=the drive traverse with the speed in P0108)
     Bit9 : BOOL ;	//JOG2 (1=the drive traverse with the speed in P0109)
     Bit10 : BOOL ;	//Control requested (Should be set 1 when ZSW1.9=1)
     Bit11 : BOOL ;	//Stop referencing (1=start the referencing point approach)
     Bit12 : BOOL ;	//Opening the holding brake for test purposes
     Bit13 : BOOL ;	//External block change (With a edge the external block changing is initiated)
     Bit14 : BOOL ;	//Reserved
     Bit15 : BOOL ;	//Request passive referencing
     Bit0 : BOOL ;	//OFF1 (1=enable)
     Bit1 : BOOL ;	//OFF2 (1=enable)
     Bit2 : BOOL ;	//OFF3 (1=enable)
     Bit3 : BOOL ;	//Pulse inhibit (0=the motor stop for inertia)
     Bit4 : BOOL ;	//Reject travel task (0=stop the motor and delete the distance to go)
     Bit5 : BOOL ;	//Intermediate stop (0=stop the motor but the process is continued with 0/1 edge)
     Bit6 : BOOL ;	//Activate travel task (With a edge the traversing block selected is started)
     Bit7 : BOOL ;	//Reset the fault memory (1=Reset the fault memory)
    END_STRUCT ;
    SatzAnw : STRUCT 	//Block selection control word
     Bit8 : BOOL ;	//Reserved
     Bit9 : BOOL ;	//Reserved
     Bit10 : BOOL ;	//Reserved
     Bit11 : BOOL ;	//Reserved
     Bit12 : BOOL ;	//Reserved
     Bit13 : BOOL ;	//Reserved
     Bit14 : BOOL ;	//Reserved
     Bit15 : BOOL ;	//Activate MDI
     Bit0 : BOOL ;	//Bit 0 block selection
     Bit1 : BOOL ;	//Bit 1 block selection
     Bit2 : BOOL ;	//Bit 2 block selection
     Bit3 : BOOL ;	//Bit 3 block selection
     Bit4 : BOOL ;	//Bit 4 block selection
     Bit5 : BOOL ;	//Bit 5 block selection
     Bit6 : BOOL ;	//Reserved
     Bit7 : BOOL ;	//Reserved
    END_STRUCT ;
    PosStw : STRUCT 	//Position control word
     Bit8 : BOOL ;	//Reserved
     Bit9 : BOOL ;	//Reserved
     Bit10 : BOOL ;	//Reserved
     Bit11 : BOOL ;	//Reserved
     Bit12 : BOOL ;	//Reserved
     Bit13 : BOOL ;	//Reserved
     Bit14 : BOOL ;	//Reserved
     Bit15 : BOOL ;	//Reserved
     Bit0 : BOOL ;	//Tracking operation (1=select tracking operation)
     Bit1 : BOOL ;	//Set reference point (0/1 edge=P0160 is assigned as actual value)
     Bit2 : BOOL ;	//Reference cams (1=the axis is located at reference cam)
     Bit3 : BOOL ;	//Fixed endstop (1=fixed endstop reached)
     Bit4 : BOOL ;	//Activate the coupling (0/1 edge=activate coupling set via P0410)
     BIt5 : BOOL ;	//Incremental jogging (1=jog in velocity and increments)
     Bit6 : BOOL ;	//Activate Teach-In (0/1=Activate Teach-In; 1/0=Reset Teach-In)
     Bit7 : BOOL ;	//Invert the angular encoder input
    END_STRUCT ;
    STW2 : STRUCT 	//Control word 2
     Bit8 : BOOL ;	//Suppress fault 608
     Bit9 : BOOL ;	//n.u. (used only in the n-set mode)
     Bit10 : BOOL ;	//n.u. (used only in the n-set mode)
     Bit11 : BOOL ;	//n.u. (used only in the n-set mode)
     Bit12 : BOOL ;	//Master sign-of-life
     Bit13 : BOOL ;	//Master sign-of-life
     Bit14 : BOOL ;	//Master sign-of-life
     Bit15 : BOOL ;	//Master sign-of-life
     Bit0 : BOOL ;	//Bit 0 parameter set changeover
     Bit1 : BOOL ;	//Bit 1 parameter set changeover
     Bit2 : BOOL ;	//Bit 2 parameter set changeover
     Bit3 : BOOL ;	//First speed setpoint filter disabled
     Bit4 : BOOL ;	//Rump-function generator enabled
     Bit5 : BOOL ;	//Reserved
     Bit6 : BOOL ;	//Integrator inhibit
     Bit7 : BOOL ;	//Select parking axis
    END_STRUCT ;
    Over : INT ;	//Percentage value for the velocity override
   END_STRUCT ;
  END_STRUCT ;
  Enable : BOOL ;	//Enable the drive
  Reset_Alarms : BOOL ;	//Reset the alarms
  Reset_Axis : BOOL ;	//Stop all the movements
  Start_Inc : BOOL ;	//Start incremental movement
  Start_Abs : BOOL ;	//Start absolute movement
  Start_Rep : BOOL ;	//Start repositioning movement
  Start_Ref : BOOL ;	//Start referencing movement
  Stop : BOOL ;	//Intermediate stop movement
  Jog_Forward : BOOL ;	//Jog forward command
  Jog_Backward : BOOL ;	//Jog backward command
  STAT58 : BOOL ;	//Reserved
  STAT57 : BOOL ;	//Reserved
  STAT56 : BOOL ;	//Reserved
  STAT55 : BOOL ;	//Reserved
  STAT54 : BOOL ;	//Reserved
  STAT53 : BOOL ;	//Reserved
  Step1_Inc : BOOL ;	//Step 1 for incremental movement management
  Step2_Inc : BOOL ;	//Step 2 for incremental movement management
  Step1_Abs : BOOL ;	//Step 1 for absolute movement management
  Step2_Abs : BOOL ;	//Step 2 for absolute movement management
  STAT36 : BOOL ;	//Reserved
  STAT35 : BOOL ;	//Reserved
  STAT34 : BOOL ;	//Reserved
  STAT33 : BOOL ;	//Reserved
  InZeroPosition : BOOL ;	//Axis in "zero" position
  AxisStationery : BOOL ;	//Axis stationery
  DriveOK : BOOL ;	//Drive OK
  BrakeOpen : BOOL ;	//Open holding brake request
  AxisOnHWHomeCam : BOOL ;	//Axis on hardware home cam
  AxisOnHWSwitchN : BOOL ;	//Axis on minus hardware extra-corse limit switch
  AxisOnHWSwitchP : BOOL ;	//Axis on plus hardware extra-corse limit switch
  AxisOnSWSwitchN : BOOL ;	//Axis on minus software extra-corse limit switch
  AxisOnSWSwitchP : BOOL ;	//Axis on plus software extra-corse limit switch
  STAT69 : BOOL ;	//Reserved
  STAT67 : BOOL ;	//Reserved
  STAT66 : BOOL ;	//Reserved
  STAT65 : BOOL ;	//Reserved
  STAT64 : BOOL ;	//Reserved
  STAT63 : BOOL ;	//Reserved
  STAT70 : BOOL ;	//Reserved
  Aux1 : BOOL ;	//Auxiliary for edge management
  Aux2 : BOOL ;	//Auxiliary for edge management
  Aux3 : BOOL ;	//Auxiliary for edge management
  Aux4 : BOOL ;	//Auxiliary for edge management
  Aux5 : BOOL ;	//Auxiliary for edge management
  Aux6 : BOOL ;	//Auxiliary for edge management
  Aux7 : BOOL ;	//Auxiliary for edge management
  Aux8 : BOOL ;	//Auxiliary for edge management
  Target_Inc : DINT ;	//Target for the incremental movement
  Target_Abs : DINT ;	//Target for the absolute movement
  DistanceToGo_Abs : DINT ;	//Difference between actual and new position
  Override : INT ;	//Percentage value for the velocity override
  ActualPosition : DINT ;	//Actual position value
END_VAR
VAR_TEMP
  tempAR1 : DWORD ;
  tempAR2 : DWORD ;
  tempSRC : ANY ;
  tempDST : ANY ;
  tempDWORD_1 : DWORD ;
  tempWORD_1 : WORD ;
  tempINT : INT ;
  tempDWORD_2 : DWORD ;
END_VAR
BEGIN
NETWORK
TITLE = Mapping of the inputs
      L     #IO_LAddr;
      SLD   3;
      T     #tempDWORD_1;
      L     P##In_Profibus;
      T     #tempDWORD_2;
      L     11;
NXT1: T     #tempINT;
      L     PIW [#tempDWORD_1];
      T     DIW [#tempDWORD_2];
      L     #tempDWORD_1;
      L     P#2.0;
      +D;
      T     #tempDWORD_1;
      L     #tempDWORD_2;
      L     P#2.0;
      +D;
      T     #tempDWORD_2;
      L     #tempINT;
      LOOP  NXT1;
NETWORK
TITLE = Status
//Axis stationery
      A     #In_Profibus.PZD.ZSW1.Bit13;
      AN    #In_Profibus.PZD.ZSW1.Bit12;
      =     #AxisStationery;
//Drive OK
      A     #In_Profibus.PZD.ZSW1.Bit0;
      A     #In_Profibus.PZD.ZSW1.Bit1;
      A     #In_Profibus.PZD.ZSW1.Bit2;
      AN    #In_Profibus.PZD.ZSW1.Bit3;
      A     #In_Profibus.PZD.ZSW1.Bit4;
      A     #In_Profibus.PZD.ZSW1.Bit5;
      A     #In_Profibus.PZD.ZSW1.Bit8;
      =     #DriveOK;
//Open holding brake request
      A     #In_Profibus.PZD.ZSW2.Bit5;
      =     #BrakeOpen;
//Axis on hardware home cam
      A     #In_Profibus.PZD.DIG_IN.Bit0;
      =     #AxisOnHWHomeCam;
//Axis on hardware minus extra-course limit switch
      A     #In_Profibus.PZD.DIG_IN.Bit1;
      =     #AxisOnHWSwitchN;
//Axis on hardware plus extra-course limit switch
      A     #In_Profibus.PZD.DIG_IN.Bit2;
      =     #AxisOnHWSwitchP;
//Axis on software minus extra-course limit switch
      A     #In_Profibus.PZD.PosZsw.Bit6;
      =     #AxisOnSWSwitchN;
//Axis on software plus extra-course limit switch
      A     #In_Profibus.PZD.PosZsw.Bit7;
      =     #AxisOnSWSwitchP;
//Actual position value
      L     #In_Profibus.PZD.XretrP;
      T     #ActualPosition;
NETWORK
TITLE = Commands
//Enable the drive
      A     #Enable;
      =     #Out_Profibus.PZD.STW1.Bit0;
      =     #Out_Profibus.PZD.STW1.Bit1;
      =     #Out_Profibus.PZD.STW1.Bit2;
      A     "On";
      =     #Out_Profibus.PZD.STW1.Bit3;
//Erase all the movements
      O     #Reset_Axis;
      O     #In_Profibus.PZD.ZSW1.Bit3;
      ON    #In_Profibus.PZD.ZSW1.Bit8;
      R     #Start_Inc;
      R     #Step1_Inc;
      R     #Step2_Inc;
      R     #Start_Abs;
      R     #Step1_Abs;
      R     #Step2_Abs;
      R     #Start_Rep;
      R     #Start_Ref;
      R     #Out_Profibus.PZD.STW1.Bit11;
      R     #Out_Profibus.PZD.STW1.Bit6;
//Stop the axis and erase the distance to go
      AN    #Reset_Axis;
      =     #Out_Profibus.PZD.STW1.Bit4;
//Intermediate stop the axis (the movement continued with a 0/1 edge)
      AN    #Stop;
      =     #Out_Profibus.PZD.STW1.Bit5;
//Reset alarms
      A     #Reset_Alarms;
      =     #Out_Profibus.PZD.STW1.Bit7;
//Control request (611U<->PLC communication)
      A     #In_Profibus.PZD.ZSW1.Bit9;
      =     #Out_Profibus.PZD.STW1.Bit10;
//Velocity override
      L     #Override;
      T     #Out_Profibus.PZD.Over;
NETWORK
TITLE = Movement in incremental mode
//Reset the incremental movement if the axis is the distance to go is minus then 0,05mm
      A     #Start_Inc;
      A(;
      L     #Target_Inc;
      L     50;
      <D;
      );
      A(;
      L     #Target_Inc;
      L     -50;
      >D;
      );
      R     #Start_Inc;
//Select the travel block (Block number 2=000010)
      A     #Start_Inc;
      R     #Out_Profibus.PZD.SatzAnw.Bit0;
      S     #Out_Profibus.PZD.SatzAnw.Bit1;
      R     #Out_Profibus.PZD.SatzAnw.Bit2;
      R     #Out_Profibus.PZD.SatzAnw.Bit3;
      R     #Out_Profibus.PZD.SatzAnw.Bit4;
      R     #Out_Profibus.PZD.SatzAnw.Bit5;
//Load the new position of the travel block
      A     #Start_Inc;
      AN    #Step1_Inc;
      AN    #Step2_Inc;
      S     #Step1_Inc;
      JCN   L001;
      L     #Target_Inc;
      T     #Out_Profibus.PKW.PWE;
      L     W#16#8051;
      T     #Out_Profibus.PKW.PKE;
      L     2;
      T     #Out_Profibus.PKW.IND;
L001: NOP   0;
//Check if the 611U received the change
      A     #Start_Inc;
      A     #Step1_Inc;
      AN    #Step2_Inc;
      A(;
      L     #Out_Profibus.PKW.PWE;
      L     #In_Profibus.PKW.PWE;
      ==D;
      );
      A(;
      L     W#16#5051;
      L     #In_Profibus.PKW.PKE;
      ==I;
      );
      A(;
      L     #Out_Profibus.PKW.IND;
      L     #In_Profibus.PKW.IND;
      ==I;
      );
      S     #Step2_Inc;
//Start travel task
      A     #Start_Inc;
      A     #Step1_Inc;
      A     #Step2_Inc;
      A(;
      L     #Target_Inc;
      L     #In_Profibus.PKW.PWE;
      ==D;
      );
//UN    #In_Profibus.PZD.AktSatz.Bit0
//U     #In_Profibus.PZD.AktSatz.Bit1
//UN    #In_Profibus.PZD.AktSatz.Bit2
//UN    #In_Profibus.PZD.AktSatz.Bit3
//UN    #In_Profibus.PZD.AktSatz.Bit4
//UN    #In_Profibus.PZD.AktSatz.Bit5
      AN    #Out_Profibus.PZD.STW1.Bit6;
      S     #Out_Profibus.PZD.STW1.Bit6;
      JCN   L002;
      L     0;
      T     #Out_Profibus.PKW.PKE;
      T     #Out_Profibus.PKW.IND;
      T     #Out_Profibus.PKW.PWE;
L002: NOP   0;
//End incremental movement
      A     #In_Profibus.PZD.ZSW1.Bit10;
      FP    #Aux1;
      A     #Start_Inc;
      A     #Step1_Inc;
      A     #Step2_Inc;
      A     #Out_Profibus.PZD.STW1.Bit6;
      R     #Out_Profibus.PZD.STW1.Bit6;
      R     #Start_Inc;
      R     #Step1_Inc;
      R     #Step2_Inc;
NETWORK
TITLE = Movement in absolute mode
//Movement not necessary if the axis is just in position  
      A     #Start_Abs;
      AN    #Step1_Abs;
      AN    #Step2_Abs;
      JCN   L004;
//Calculate the difference between the actual position and new position
      L     #Target_Abs;
      L     #In_Profibus.PZD.XretrP;
      -D;
      T     #DistanceToGo_Abs;
      L     0;
      <D;
      JCN   L003;
      L     #DistanceToGo_Abs;
      NEGD;
      T     #DistanceToGo_Abs;
L003: NOP   0;
      A(;
      L     #DistanceToGo_Abs;
      L     99;
      <=D;
      );
      R     #Start_Abs;
L004: NOP   0;
//Select the travel block (Block number 0=000000)
      A     #Start_Abs;
      R     #Out_Profibus.PZD.SatzAnw.Bit0;
      R     #Out_Profibus.PZD.SatzAnw.Bit1;
      R     #Out_Profibus.PZD.SatzAnw.Bit2;
      R     #Out_Profibus.PZD.SatzAnw.Bit3;
      R     #Out_Profibus.PZD.SatzAnw.Bit4;
      R     #Out_Profibus.PZD.SatzAnw.Bit5;
//Load the new position of the travel block
      A     #Start_Abs;
      AN    #Step1_Abs;
      AN    #Step2_Abs;
      S     #Step1_Abs;
      JCN   L005;
      L     #Target_Abs;
      T     #Out_Profibus.PKW.PWE;
      L     W#16#8051;
      T     #Out_Profibus.PKW.PKE;
      L     0;
      T     #Out_Profibus.PKW.IND;
L005: NOP   0;
//Check if the 611U received the change
      A     #Start_Abs;
      A     #Step1_Abs;
      AN    #Step2_Abs;
      A(;
      L     #Out_Profibus.PKW.PWE;
      L     #In_Profibus.PKW.PWE;
      ==D;
      );
      A(;
      L     W#16#5051;
      L     #In_Profibus.PKW.PKE;
      ==I;
      );
      A(;
      L     #Out_Profibus.PKW.IND;
      L     #In_Profibus.PKW.IND;
      ==I;
      );
      S     #Step2_Abs;
//Start travel task
      A     #Start_Abs;
      A     #Step1_Abs;
      A     #Step2_Abs;
      A(;
      L     #Target_Abs;
      L     #In_Profibus.PKW.PWE;
      ==D;
      );
      AN    #In_Profibus.PZD.AktSatz.Bit0;
      AN    #In_Profibus.PZD.AktSatz.Bit1;
      AN    #In_Profibus.PZD.AktSatz.Bit2;
      AN    #In_Profibus.PZD.AktSatz.Bit3;
      AN    #In_Profibus.PZD.AktSatz.Bit4;
      AN    #In_Profibus.PZD.AktSatz.Bit5;
      AN    #Out_Profibus.PZD.STW1.Bit6;
      S     #Out_Profibus.PZD.STW1.Bit6;
      JCN   L006;
      L     0;
      T     #Out_Profibus.PKW.PKE;
      T     #Out_Profibus.PKW.IND;
      T     #Out_Profibus.PKW.PWE;
L006: NOP   0;
//End absolute movement
      A     #In_Profibus.PZD.ZSW1.Bit10;
      FP    #Aux2;
      A     #Start_Abs;
      A     #Step1_Abs;
      A     #Step2_Abs;
      A     #Out_Profibus.PZD.STW1.Bit6;
      R     #Out_Profibus.PZD.STW1.Bit6;
      R     #Start_Abs;
      R     #Step1_Abs;
      R     #Step2_Abs;
NETWORK
TITLE = Repositioning management
//Movement not necessary if the axis is just in position  
      A     #Start_Rep;
      FP    #Aux3;
      A     #InZeroPosition;
      R     #Start_Rep;
//Select the travel block (Block number 1=000001)
      A     #Start_Rep;
      S     #Out_Profibus.PZD.SatzAnw.Bit0;
      R     #Out_Profibus.PZD.SatzAnw.Bit1;
      R     #Out_Profibus.PZD.SatzAnw.Bit2;
      R     #Out_Profibus.PZD.SatzAnw.Bit3;
      R     #Out_Profibus.PZD.SatzAnw.Bit4;
      R     #Out_Profibus.PZD.SatzAnw.Bit5;
//Start travel task
      A     #Start_Rep;
      A     #In_Profibus.PZD.AktSatz.Bit0;
      AN    #In_Profibus.PZD.AktSatz.Bit1;
      AN    #In_Profibus.PZD.AktSatz.Bit2;
      AN    #In_Profibus.PZD.AktSatz.Bit3;
      AN    #In_Profibus.PZD.AktSatz.Bit4;
      AN    #In_Profibus.PZD.AktSatz.Bit5;
      AN    #Out_Profibus.PZD.STW1.Bit6;
      S     #Out_Profibus.PZD.STW1.Bit6;
//End repositioning
      A     #In_Profibus.PZD.ZSW1.Bit10;
      FP    #Aux4;
      A     #Start_Rep;
      A     #Out_Profibus.PZD.STW1.Bit6;
      R     #Out_Profibus.PZD.STW1.Bit6;
      R     #Start_Rep;
NETWORK
TITLE = Jog management
//Jog forward
      A     #Jog_Forward;
      A     #In_Profibus.PZD.ZSW1.Bit11;
      AN    #In_Profibus.PZD.PosZsw.Bit7;
      =     #Out_Profibus.PZD.STW1.Bit9;
//Jog backward
      A     #Jog_Backward;
      A     #In_Profibus.PZD.ZSW1.Bit11;
      AN    #In_Profibus.PZD.PosZsw.Bit6;
      =     #Out_Profibus.PZD.STW1.Bit8;
NETWORK
TITLE = Referencing management
//Start the referencing point approach
      A     #Start_Ref;
      FP    #Aux5;
      S     #Out_Profibus.PZD.STW1.Bit11;
//End of referencing point approch
      A     #In_Profibus.PZD.ZSW1.Bit11;
      FP    #Aux6;
      R     #Out_Profibus.PZD.STW1.Bit11;
      R     #Start_Ref;
NETWORK
TITLE = Mapping of the outputs
      L     #IO_LAddr;
      SLD   3;
      T     #tempDWORD_1;
      L     P##Out_Profibus;
      T     #tempDWORD_2;
      L     9;
NXT3: T     #tempINT;
      L     DIW [#tempDWORD_2];
      T     PQW [#tempDWORD_1];
      L     #tempDWORD_1;
      L     P#2.0;
      +D;
      T     #tempDWORD_1;
      L     #tempDWORD_2;
      L     P#2.0;
      +D;
      T     #tempDWORD_2;
      L     #tempINT;
      LOOP  NXT3;
END_FUNCTION_BLOCK

FUNCTION_BLOCK "BALLUFF"	// FB 20
TITLE = BALLUFF Reader/Writer management
VERSION : 0.1
VAR_INPUT
  IO_LAddr : INT ;
END_VAR
VAR
  InputBuffer : STRUCT
   CP : BOOL ;	//Codetag present
   AA : BOOL ;	//Command started
   AE : BOOL ;	//Command finished without error
   AF : BOOL ;	//Command finished with error
   KN : BOOL ;	//Header number
   TO : BOOL ;	//Toggle-bit Out
   HF : BOOL ;	//Head error
   BB : BOOL ;	//Ready
   ErrorCode : BYTE ;
   Data1 : BYTE ;
   Data2 : BYTE ;
   Data3 : BYTE ;
   Data4 : BYTE ;
  END_STRUCT ;
  OutputBuffer : STRUCT
   AV : BOOL ;	//Command
   Reserved1 : BOOL ;
   GR : BOOL ;	//Ground state
   Reserved2 : BOOL ;
   HD : BOOL ;	//Head direct
   Reserved3 : BOOL ;
   TI : BOOL ;	//Toggle-bit in
   CT : BOOL ;	//Codetag type
   Command : BYTE ;
   StartAddress_L : BYTE ;
   StartAddress_H : BYTE ;
   NoBytes_L : BYTE ;
   NoBytes_H : BYTE ;
  END_STRUCT ;
  Testa1 : STRUCT
   Lettura_Start : BOOL ;	//1=start read job
   Lettura_OK : BOOL ;	//1=read job ended without error
   Lettura_NOK : BOOL ;	//1=read job ended with error
   Lettura_Step1 : BOOL ;	//Aux for read job cycle
   Lettura_Step2 : BOOL ;	//Aux for read job cycle
   Lettura_Step3 : BOOL ;	//Aux for read job cycle
   Lettura_Step4 : BOOL ;	//Aux for read job cycle
   Lettura_Step5 : BOOL ;	//Aux for read job cycle
   Scrittura_Start : BOOL ;	//1=start write job
   Scrittura_OK : BOOL ;	//1=write job ended without error
   Scrittura_NOK : BOOL ;	//1=write job ended with error
   Scrittura_Step1 : BOOL ;	//Aux for write job cycle
   Scrittura_Step2 : BOOL ;	//Aux for write job cycle
   Scrittura_Step3 : BOOL ;	//Aux for write job cycle
   Scrittura_Step4 : BOOL ;	//Aux for write job cycle
   Scrittura_Step5 : BOOL ;	//Aux for write job cycle
   ValoreLetto : BYTE ;	//Data readed
   ValoreDaScrivere : BYTE ;	//Data to write
   Seconds : BYTE ;	//Number of seconds of activity
  END_STRUCT ;
  Testa2 : STRUCT
   Lettura_Start : BOOL ;	//1=start read job
   Lettura_OK : BOOL ;	//1=read job ended without error
   Lettura_NOK : BOOL ;	//1=read job ended with error
   Lettura_Step1 : BOOL ;	//Aux for read job cycle
   Lettura_Step2 : BOOL ;	//Aux for read job cycle
   Lettura_Step3 : BOOL ;	//Aux for read job cycle
   Lettura_Step4 : BOOL ;	//Aux for read job cycle
   Lettura_Step5 : BOOL ;	//Aux for read job cycle
   Scrittura_Start : BOOL ;	//1=start write job
   Scrittura_OK : BOOL ;	//1=write job ended without error
   Scrittura_NOK : BOOL ;	//1=write job ended with error
   Scrittura_Step1 : BOOL ;	//Aux for write job cycle
   Scrittura_Step2 : BOOL ;	//Aux for write job cycle
   Scrittura_Step3 : BOOL ;	//Aux for write job cycle
   Scrittura_Step4 : BOOL ;	//Aux for write job cycle
   Scrittura_Step5 : BOOL ;	//Aux for write job cycle
   ValoreLetto : BYTE ;	//Data readed
   ValoreDaScrivere : BYTE ;	//Data to write
   Seconds : BYTE ;	//Number of seconds of activity
  END_STRUCT ;
END_VAR
VAR_TEMP
  tempAR1 : DWORD ;
  tempAR2 : DWORD ;
  tempSRC : ANY ;
  tempDST : ANY ;
  tempDWORD_1 : DWORD ;
  tempWORD_1 : WORD ;
  tempINT : INT ;
  tempBYTE1 : BYTE ;
  tempBYTE2 : BYTE ;
END_VAR
BEGIN
NETWORK
TITLE = Mapping of the inputs
//Save registry value
      TAR1  #tempAR1;
      TAR2  #tempAR2;
//Creation of a pointer to the source area
      LAR1  P##tempSRC;	//Load initial address of source pointer in AR1
      L     B#16#10;	//Load the ID for the ANY type
      T     LB [AR1,P#0.0];
      L     B#16#2;	//2=type of data is BYTE
      T     LB [AR1,P#1.0];
      L     6;	//Number of bytess to transfer
      T     LW [AR1,P#2.0];
      L     0;	//Type of data memory
      T     LW [AR1,P#4.0];
      L     DIW 0;
      SLD   3;
      L     P#I 0.0;
      +D;
      T     LD [AR1,P#6.0];
//Creation of a pointer to the target area
      LAR1  P##tempDST;	//Load initial address of destination pointer in AR1
      L     B#16#10;	//Load the ID for the ANY type
      T     LB [AR1,P#0.0];
      L     B#16#2;	//2=type of data is BYTE
      T     LB [AR1,P#1.0];
      L     6;	//Number of bytes to receive
      T     LW [AR1,P#2.0];
      L     0;	//Type of data memory
      T     LW [AR1,P#4.0];
      L     P##InputBuffer;
      T     LD [AR1,P#6.0];
//Trasfering data
      CALL  "BLKMOV" (
           SRCBLK                   := #tempSRC,
           RET_VAL                  := #tempINT,
           DSTBLK                   := #tempDST);
//Load saved registry value
      LAR1  #tempAR1;
      LAR2  #tempAR2;
NETWORK
TITLE = Mapping of the outputs
//Save registry value
      TAR1  #tempAR1;
      TAR2  #tempAR2;
//Creation of a pointer to the source area
      LAR1  P##tempSRC;	//Load initial address of source pointer in AR1
      L     B#16#10;	//Load the ID for the ANY type
      T     LB [AR1,P#0.0];
      L     B#16#2;	//2=type of data is BYTE
      T     LB [AR1,P#1.0];
      L     6;	//Number of bytess to transfer
      T     LW [AR1,P#2.0];
      L     0;	//Type of data memory
      T     LW [AR1,P#4.0];
      L     DIW 0;
      SLD   3;
      L     P#Q 0.0;
      +D;
      T     LD [AR1,P#6.0];
//Creation of a pointer to the target area
      LAR1  P##tempDST;	//Load initial address of destination pointer in AR1
      L     B#16#10;	//Load the ID for the ANY type
      T     LB [AR1,P#0.0];
      L     B#16#2;	//2=type of data is BYTE
      T     LB [AR1,P#1.0];
      L     6;	//Number of bytes to receive
      T     LW [AR1,P#2.0];
      L     0;	//Type of data memory
      T     LW [AR1,P#4.0];
      L     P##OutputBuffer;
      T     LD [AR1,P#6.0];
//Trasfering data
      CALL  "BLKMOV" (
           SRCBLK                   := #tempSRC,
           RET_VAL                  := #tempINT,
           DSTBLK                   := #tempDST);
//Load saved registry value
      LAR1  #tempAR1;
      LAR2  #tempAR2;
NETWORK
TITLE = Read job of header 1
      A     DIX 14.3;
      A     "Clock_P";
      JCN   L006;
      L     DIB 18;
      L     1;
      +I;
      T     DIB 18;
L006: NOP   0;
//Select the header
      A     DIX 14.0;
      AN    DIX 15.0;
//UN    #Testa2.Lettura_Start
//UN    #Testa2.Scrittura_Start
      AN    DIX 14.3;
      S     DIX 14.3;
      R     DIX 8.4;
      JCN   L005;
      L     0;
      T     DIB 18;
L005: NOP   0;
//Check the header selected
      A     DIX 14.0;
      A     DIX 14.3;
      AN    DIX 2.4;
      AN    DIX 14.4;
      S     DIX 14.4;
//Start reading job
      A     DIX 14.0;
      A     DIX 14.4;
      A     DIX 2.7;
      A     DIX 2.0;
      AN    DIX 14.5;
      S     DIX 14.5;
      R     DIX 14.1;
      R     DIX 14.2;
      S     DIX 8.0;
      R     DIX 8.7;
      JC    L001;
      JU    L004;
L001: NOP   0;
      L     0;
      T     DIB 10;
      T     DIB 11;
      T     DIB 13;
      L     1;
      T     DIB 12;
      L     1;
      T     DIB 9;
L004: NOP   0;
//Read job ended with error
      A     DIX 14.0;
      A     DIX 14.5;
      A     DIX 2.1;
      A     DIX 2.3;
      O;
      A(;
      L     DIB 18;
      L     10;
      >=I;
      );
      R     DIX 14.3;
      R     DIX 14.4;
      R     DIX 14.5;
      R     DIX 8.0;
      R     DIX 14.0;
      S     DIX 14.2;
      JCN   L007;
      L     0;
      T     DIB 18;
L007: NOP   0;
//Read job ended without error
      A     DIX 14.0;
      A     DIX 14.5;
      A     DIX 2.1;
      A     DIX 2.2;
      R     DIX 14.3;
      R     DIX 14.4;
      R     DIX 14.5;
      R     DIX 8.0;
      R     DIX 14.0;
      S     DIX 14.1;
      JC    L002;
      JU    L003;
L002: L     DIB 3;
//T     #tempBYTE1
//L     #InputBuffer.Data1
//T     #tempBYTE2
//L     LW    36
      T     DIB 16;
L003: NOP   0;
NETWORK
TITLE = Write job of header 1
      A     DIX 15.3;
      A     "Clock_P";
      JCN   L018;
      L     DIB 18;
      L     1;
      +I;
      T     DIB 18;
L018: NOP   0;
//Select the header
      A     DIX 15.0;
      AN    DIX 14.0;
//UN    #Testa2.Lettura_Start
//UN    #Testa2.Scrittura_Start
      AN    DIX 15.3;
      S     DIX 15.3;
      R     DIX 8.4;
      JCN   L015;
      L     0;
      T     DIB 18;
L015: NOP   0;
//Check the header selected
      A     DIX 15.0;
      A     DIX 15.3;
      AN    DIX 2.4;
      AN    DIX 15.4;
      S     DIX 15.4;
//Start writing job
      A     DIX 15.0;
      A     DIX 15.4;
      A     DIX 2.7;
      A     DIX 2.0;
      AN    DIX 15.5;
      S     DIX 15.5;
      R     DIX 15.1;
      R     DIX 15.2;
      S     DIX 8.0;
      R     DIX 8.7;
      JC    L011;
      JU    L012;
L011: NOP   0;
      L     0;
      T     DIB 10;
      T     DIB 11;
      T     DIB 13;
      L     1;
      T     DIB 12;
      L     2;
      T     DIB 9;
L012: NOP   0;
//Confirm write job in course
      A     DIX 15.0;
      A     DIX 15.5;
      A     DIX 2.1;
      A     DIX 2.5;
      AN    DIX 15.6;
      S     DIX 15.6;
      S     DIX 8.6;
      JC    L016;
      JU    L017;
L016: NOP   0;
      L     DIB 17;
//T     LW    36
//L     #tempBYTE1
      T     DIB 9;
//L     #tempBYTE2
//T     #OutputBuffer.StartAddress_L
L017: NOP   0;
//Write job ended with error
      A     DIX 15.0;
      A     DIX 15.6;
      A     DIX 2.1;
      A     DIX 2.3;
      O;
      A(;
      L     DIB 18;
      L     10;
      >=I;
      );
      R     DIX 15.3;
      R     DIX 15.4;
      R     DIX 15.5;
      R     DIX 15.6;
      R     DIX 8.0;
      R     DIX 8.6;
      R     DIX 15.0;
      S     DIX 15.2;
      JCN   L019;
      L     0;
      T     DIB 18;
L019: NOP   0;
//Write job ended without error
      A     DIX 15.0;
      A     DIX 15.6;
      A     DIX 2.1;
      A     DIX 2.2;
      R     DIX 15.3;
      R     DIX 15.4;
      R     DIX 15.5;
      R     DIX 15.6;
      R     DIX 8.0;
      R     DIX 8.6;
      R     DIX 15.0;
      S     DIX 15.1;
NETWORK
TITLE = Read job of header 2
      A     DIX 20.3;
      A     "Clock_P";
      JCN   L026;
      L     DIB 24;
      L     1;
      +I;
      T     DIB 24;
L026: NOP   0;
//Select the header
      A     DIX 20.0;
      AN    DIX 21.0;
      AN    DIX 14.0;
      AN    DIX 15.0;
      AN    DIX 20.3;
      S     DIX 20.3;
      S     DIX 8.4;
      JCN   L025;
      L     0;
      T     DIB 24;
L025: NOP   0;
//Check the header selected
      A     DIX 20.0;
      A     DIX 20.3;
      A     DIX 2.4;
      AN    DIX 20.4;
      S     DIX 20.4;
//Start reading job
      A     DIX 20.0;
      A     DIX 20.4;
      A     DIX 2.7;
      A     DIX 2.0;
      AN    DIX 20.5;
      S     DIX 20.5;
      R     DIX 20.1;
      R     DIX 20.2;
      S     DIX 8.0;
      R     DIX 8.7;
      JC    L021;
      JU    L024;
L021: NOP   0;
      L     0;
      T     DIB 10;
      T     DIB 11;
      T     DIB 13;
      L     1;
      T     DIB 12;
      L     1;
      T     DIB 9;
L024: NOP   0;
//Read job ended with error
      A     DIX 20.0;
      A     DIX 20.5;
      A     DIX 2.1;
      A     DIX 2.3;
      O;
      A(;
      L     DIB 24;
      L     10;
      >=I;
      );
      R     DIX 20.3;
      R     DIX 20.4;
      R     DIX 20.5;
      R     DIX 8.0;
      R     DIX 20.0;
      S     DIX 20.2;
      JCN   L027;
      L     0;
      T     DIB 24;
L027: NOP   0;
//Read job ended without error
      A     DIX 20.0;
      A     DIX 20.5;
      A     DIX 2.1;
      A     DIX 2.2;
      R     DIX 20.3;
      R     DIX 20.4;
      R     DIX 20.5;
      R     DIX 8.0;
      R     DIX 20.0;
      S     DIX 20.1;
      JC    L022;
      JU    L023;
L022: L     DIB 3;
//T     #tempBYTE1
//L     #InputBuffer.Data1
//T     #tempBYTE2
//L     LW    36
      T     DIB 22;
L023: NOP   0;
NETWORK
TITLE = Write job of header 2
      A     DIX 21.3;
      A     "Clock_P";
      JCN   L038;
      L     DIB 24;
      L     1;
      +I;
      T     DIB 24;
L038: NOP   0;
//Select the header
      A     DIX 21.0;
      AN    DIX 20.0;
      AN    DIX 14.0;
      AN    DIX 15.0;
      AN    DIX 21.3;
      S     DIX 21.3;
      S     DIX 8.4;
      JCN   L035;
      L     0;
      T     DIB 24;
L035: NOP   0;
//Check the header selected
      A     DIX 21.0;
      A     DIX 21.3;
      A     DIX 2.4;
      AN    DIX 21.4;
      S     DIX 21.4;
//Start writing job
      A     DIX 21.0;
      A     DIX 21.4;
      A     DIX 2.7;
      A     DIX 2.0;
      AN    DIX 21.5;
      S     DIX 21.5;
      R     DIX 21.1;
      R     DIX 21.2;
      S     DIX 8.0;
      R     DIX 8.7;
      JC    L031;
      JU    L032;
L031: NOP   0;
      L     0;
      T     DIB 10;
      T     DIB 11;
      T     DIB 13;
      L     1;
      T     DIB 12;
      L     2;
      T     DIB 9;
L032: NOP   0;
//Confirm write job in course
      A     DIX 21.0;
      A     DIX 21.5;
      A     DIX 2.1;
      A     DIX 2.5;
      AN    DIX 21.6;
      S     DIX 21.6;
      S     DIX 8.6;
      JC    L036;
      JU    L037;
L036: NOP   0;
      L     DIB 23;
//T     LW    36
//L     #tempBYTE1
      T     DIB 9;
//L     #tempBYTE2
//T     #OutputBuffer.StartAddress_L
L037: NOP   0;
//Write job ended with error
      A     DIX 21.0;
      A     DIX 21.6;
      A     DIX 2.1;
      A     DIX 2.3;
      O;
      A(;
      L     DIB 24;
      L     10;
      >=I;
      );
      R     DIX 21.3;
      R     DIX 21.4;
      R     DIX 21.5;
      R     DIX 21.6;
      R     DIX 8.0;
      R     DIX 8.6;
      R     DIX 21.0;
      S     DIX 21.2;
      JCN   L039;
      L     0;
      T     DIB 24;
L039: NOP   0;
//Write job ended without error
      A     DIX 21.0;
      A     DIX 21.6;
      A     DIX 2.1;
      A     DIX 2.2;
      R     DIX 21.3;
      R     DIX 21.4;
      R     DIX 21.5;
      R     DIX 21.6;
      R     DIX 8.0;
      R     DIX 8.6;
      R     DIX 21.0;
      S     DIX 21.1;
NETWORK
TITLE = Mapping of the outputs
//Save registry value
      TAR1  #tempAR1;
      TAR2  #tempAR2;
//Creation of a pointer to the source area
      LAR1  P##tempSRC;	//Load initial address of source pointer in AR1
      L     B#16#10;	//Load the ID for the ANY type
      T     LB [AR1,P#0.0];
      L     B#16#2;	//2=type of data is BYTE
      T     LB [AR1,P#1.0];
      L     6;	//Number of bytess to transfer
      T     LW [AR1,P#2.0];
      L     0;	//Type of data memory
      T     LW [AR1,P#4.0];
      L     P##OutputBuffer;
      T     LD [AR1,P#6.0];
//Creation of a pointer to the target area
      LAR1  P##tempDST;	//Load initial address of destination pointer in AR1
      L     B#16#10;	//Load the ID for the ANY type
      T     LB [AR1,P#0.0];
      L     B#16#2;	//2=type of data is BYTE
      T     LB [AR1,P#1.0];
      L     6;	//Number of bytes to receive
      T     LW [AR1,P#2.0];
      L     0;	//Type of data memory
      T     LW [AR1,P#4.0];
      L     DIW 0;
      SLD   3;
      L     P#Q 0.0;
      +D;
      T     LD [AR1,P#6.0];
//Trasfering data
      CALL  "BLKMOV" (
           SRCBLK                   := #tempSRC,
           RET_VAL                  := #tempINT,
           DSTBLK                   := #tempDST);
//Load saved registry value
      LAR1  #tempAR1;
      LAR2  #tempAR2;
END_FUNCTION_BLOCK

FUNCTION_BLOCK "FB24 - Gestione Mov Assi"	// FB 24
TITLE = GESTIONE ASSI STAZIONE OP60
VERSION : 0.1
VAR_INPUT
  INDIRIZZO_INIZIALE_E_A : DINT ;	//INDIRIZZO INIZIALE I/O (VEDI CONFIGURAZIONE HARDWARE)
  OK_FOR_COMMANDS : BOOL ;	//TUTTO PRONTO PER I COMANDI
  RESET_ALLARMI : BOOL ;	//1=RESET ALLARMI AZIONAMENTO
  STOP : BOOL ;	//0=STOP DI TUTTI I MOVIMENTI
  TARGET_POSIZIONE : DINT ;	//TARGET DI POSIZIONAMENTO ASSOLUTO
  TARGET_INCREMENTALE : DINT ;	//SPOSTAMENTO IN MODO INCREMENTALE
  OVERRIDE : INT ;	//OVVERIDE DI VELOCITA'
  JOG_PIU : BOOL ;	//COMANDO JOG PIU'
  JOG_MENO : BOOL ;	//COMANDO JOG MENO
  IN_PKE : WORD ;
  IN_IND : WORD ;
  IN_PWE : DINT ;
  ASSE_SU_HOME : BOOL ;	//ASSE GIA' SU POSIZIONE DI HOME
END_VAR
VAR_OUTPUT
  OUT_PKE : WORD ;
  OUT_IND : WORD ;
  OUT_PWE : DINT ;
  POSIZIONE_ATTUALE : DINT ;
  POSIZIONE_RAGGIUNTA : BOOL ;	//POSIZIONAMENTO ULTIMATO
  HOME_OK : BOOL ;	//1=ASSE RIFERITO
  RIPOSIZIONAMENTO_OK : BOOL ;	//1=RIPOSIZIONAMENTO EFFETTUATO
  ASSE_FERMO_NO_JOB : BOOL ;	//1=ASSE FERMO E NESSUN JOB IN CORSO
  AZIONAMENTO_OK : BOOL ;	//1=AZIONAMENTO PRONTO
  AZIONAMENTO_FAULT : BOOL ;	//1=AZIONAMENTO IN ALLARME
  CAMMA_DI_RIFERIMENTO : BOOL ;	//1=ASSE SU CAMMA DI RIFERIMENTO
  OLTRECORSA_NEGATIVO : BOOL ;	//1=ASSE SU OLTRECORSA HARDWARE NEGATIVO
  OLTRECORSA_POSITIVO : BOOL ;	//1=ASSE SU OLTRECORSA HARDWARE POSITIVO
  FINECORSA_SOFTWARE_NEG : BOOL ;	//1=FINECORSA SOFTWARE NEGATIVO
  FINECORSA_SOFTWARE_POS : BOOL ;	//1=FINECORSA SOFTWARE POSITIVO
  FRENO : BOOL ;	//1=APRIRE IL FRENO DI STAZIONAMENTO
END_VAR
VAR_IN_OUT
  START_ASSOLUTO : BOOL ;	//1=START POSIZIONAMENTO ASSOLUTO
  START_INCREMENTALE : BOOL ;	//1=START POSIZIONAMENTO INCREMENTALE
  START_HOME : BOOL ;	//1=START RICERCA ZERO
  START_RIPOSIZIONAMENTO : BOOL ;	//1=START POSIZIONAMENTO SU POSIZIONE INIZIALE
END_VAR
VAR
  SCELTA_BLOCCO : WORD ;
  BLOCCO_ATTUALE : WORD ;
  INVIA_JOB1 : BOOL ;	//INVIO COMANDO DI CARICA BLOCCO ASSOLUTO
  JOB1_ULTIMATO : BOOL ;	//IL NUOVO BLOCCO DI MOVIMENTO ASSOLUTO E' STATO INVIATO
  INVIA_JOB2 : BOOL ;	//INVIO COMANDO DI CARICA BLOCCO INCREMENTALE
  JOB2_ULTIMATO : BOOL ;	//IL NUOVO BLOCCO DI MOVIMENTO INCREMENTALE E' STATO INVIATO
  GIA_IN_POSIZIONE : BOOL ;	//POSIZIONAMENTO NON NECESSARIO PER ASSE GIA' IN POSIZIONE
  PACO1 : STRUCT
   PACO1_8 : BOOL ;	//1=MARCIA A IMPULSI 1
   PACO1_9 : BOOL ;	//1=MARCIA 1 IMPULSI 2
   PACO1_10 : BOOL ;	//1=ABILITA IL COMANDO (DA METTERE A 1 QUANDO PAST1.9=1)
   PACO1_11 : BOOL ;	//1=AVVIA IL RIFERIMENTO DELL'ASSE
   PACO1_12 : BOOL ;	//RISERVATO
   PACO1_13 : BOOL ;	//1=CAMBIO BLOCCO ESTERNO
   PACO1_14 : BOOL ;	//RISERVATO
   PACO1_15 : BOOL ;	//RISERVATO
   PACO1_0 : BOOL ;	//1=INSERITO 0=DISINSERITO
   PACO1_1 : BOOL ;	//1=INSERITO 0=DISINSERITO
   PACO1_2 : BOOL ;	//1=INSERITO 0=DISINSERITO
   PACO1_3 : BOOL ;	//0=BLOCCO IMPULSI (IL MOTORE SI FERMA PER INERZIA)
   PACO1_4 : BOOL ;	//1=OK 0=STOP ASSE E CANCELLAZIONE PERCORSO RESISDUO
   PACO1_5 : BOOL ;	//1=OK 0=STOP ASSE E ULTIMAZIONE MOVIMENTO CON FRONTE 0-->1
   PACO1_6 : BOOL ;	//0-->1=ATTIVARE L'ORDINE DI SPOSTAMENTO
   PACO1_7 : BOOL ;	//1=TACITAZIONE ALLARME
  END_STRUCT ;
  PAST1 : STRUCT
   PAST1_8 : BOOL ;	//1=NESSUN ERRORE D'INSEGUIMENTO
   PAST1_9 : BOOL ;	//1=SLAVE OK E PRONTO A RICEVERE COMANDI
   PAST1_10 : BOOL ;	//1=POSIZIONE RAGGIUNTA
   PAST1_11 : BOOL ;	//1=ASSE RIFERITO
   PAST1_12 : BOOL ;	//1=POSIZIONAMENTO IN CORSO
   PAST1_13 : BOOL ;	//1=MOTORE FERMO
   PAST1_14 : BOOL ;	//RISERVATO
   PAST1_15 : BOOL ;	//RISERVATO
   PAST1_0 : BOOL ;	//1=PRONTO ALL'INSERZIONE
   PAST1_1 : BOOL ;	//1=PRONTO AL FUNZIONAMENTO
   PAST1_2 : BOOL ;	//STATO ABILITAZIONE REGOLATORE
   PAST1_3 : BOOL ;	//1=PRESEZA GUASTI
   PAST1_4 : BOOL ;	//1=DISINSERIMENTO 2 ASSENTE
   PAST1_5 : BOOL ;	//1=DISINSERIMENTO 3 ASSENTE
   PAST1_6 : BOOL ;	//1=BLOCCO ALL'INSERZIONE
   PAST1_7 : BOOL ;	//1=PRESENZA AVVISI
  END_STRUCT ;
  DIGin : STRUCT
   DIGin_8 : BOOL ;
   DIGin_9 : BOOL ;
   DIGin_10 : BOOL ;
   DIGin_11 : BOOL ;
   DIGin_12 : BOOL ;
   DIGin_13 : BOOL ;
   DIGin_14 : BOOL ;
   DIGin_15 : BOOL ;
   DIGin_0 : BOOL ;	//1=ASSE SU CAMMA DI HOME
   DIGin_1 : BOOL ;	//1=ASSE SU EXTRACORSA NEGATIVO
   DIGin_2 : BOOL ;	//1=ASSE SU EXTRACORSA POSITIVO
   DIGin_3 : BOOL ;
   DIGin_4 : BOOL ;
   DIGin_5 : BOOL ;
   DIGin_6 : BOOL ;
   DIGin_7 : BOOL ;
  END_STRUCT ;
  AUX1 : BOOL ;	//APPOGGIO PER FRONTE
  AUX2 : BOOL ;	//APPOGGIO PER FRONTE
  AUX3 : BOOL ;	//APPOGGIO PER FRONTE
  AUX4 : BOOL ;	//APPOGGIO PER FRONTE
  AUX5 : BOOL ;	//APPOGGIO PER FRONTE
  AUX6 : BOOL ;	//APPOGGIO PER FRONTE
  AUX7 : BOOL ;	//APPOGGIO PER FRONTE
  VERIFICA_SPOSTAMENTO : DINT ;	//DIFFERENZA TRA TARGET E POSIZIONE ATTUALE
  PAST2 : STRUCT
   PAST2_8 : BOOL ;	//1=TACITARE IL GUASTO 608
   PAST2_9 : BOOL ;	//1=ATTUALE MOTORE 1.SEGNALE
   PAST2_10 : BOOL ;	//1=ATTUALE MOTORE 2.SEGNALE
   PAST2_11 : BOOL ;	//1=RISERVATO
   PAST2_12 : BOOL ;
   PAST2_13 : BOOL ;
   PAST2_14 : BOOL ;
   PAST2_15 : BOOL ;
   PAST2_0 : BOOL ;
   PAST2_1 : BOOL ;
   PAST2_2 : BOOL ;
   PAST2_3 : BOOL ;	//PRIMO FILTRO DEL RIFERIMENTO ATTIVO
   PAST2_4 : BOOL ;	//BLOCCO DELL'INTEGRATORE NEL REGOLATORE DI VELOCITA'
   PAST2_5 : BOOL ;	//APRIRE IL FRENO DI STAZIONAMENTO
   PAST2_6 : BOOL ;	//BLOCCO DELL'INTEGRATORE NEL REGOLATORE DI VELOCITA'
   PAST2_7 : BOOL ;	//SCELTO L'ASSE IN PARCHEGGIO
  END_STRUCT ;
  POS_PAST : STRUCT
   POS_PAST_0 : BOOL ;	//FUNZIONAMENTO A SEGUIRE
   POS_PAST_1 : BOOL ;	//LIMITAZIONE DELLA VELOCITA' LINEARE ATTIVA
   POS_PAST_2 : BOOL ;	//C'E' IL RIFERIMENTO
   POS_PAST_3 : BOOL ;	//BIT DI FUNZIONE
   POS_PAST_4 : BOOL ;	//L'ASSE SI SPOSTA IN AVANTI
   POS_PAST_5 : BOOL ;	//L'ASSE SI SPOSTA INDIETRO
   POS_PAST_6 : BOOL ;	//FINECORSA SOFTWARE MENO
   POS_PAST_7 : BOOL ;	//FINECORSA SOFTWARE PIU'
   POS_PAST_8 : BOOL ;	//SEGNALE D'INSERZIONE DELLA CAMMA 1
   POS_PAST_9 : BOOL ;	//SEGNALE D'INSERZIONE DELLA CAMMA 2
   POS_PAST_10 : BOOL ;	//USCITA DIRETTA 1 CON IL BLOCCO DI SPOSTAMENTO
   POS_PAST_11 : BOOL ;	//USCITA DIRETTA 2 CON IL BLOCCO DI SPOSTAMENTO
   POS_PAST_12 : BOOL ;	//RISERVATO
   POS_PAST_13 : BOOL ;	//RISERVATO
   POS_PAST_14 : BOOL ;	//RISERVATO
   POS_PAST_15 : BOOL ;	//RISERVATO
  END_STRUCT ;
END_VAR
BEGIN
NETWORK
TITLE = AGGIORNAMENTO IMMAGINE INGRESSI
      L     #INDIRIZZO_INIZIALE_E_A;
      L     8;
      +I;
      SLD   3;
      T     "MD100";
      L     PIW ["MD100"];	//;PAST1
      T     DIW 52;
      L     "MD100";
      SRW   3;
      L     2;
      +D;
      SLW   3;
      T     "MD100";
//;
      L     PIW ["MD100"];	//;BLOCCO ATTUALE
      T     #BLOCCO_ATTUALE;
      L     "MD100";
      SRW   3;
      L     2;
      +D;
      SLW   3;
      T     "MD100";
//;
      L     PIW ["MD100"];	//;POS PAST
      T     DIW 64;
      L     "MD100";
      SRW   3;
      L     2;
      +D;
      SLW   3;
      T     "MD100";
//;
      L     PIW ["MD100"];	//;PAST 2
      T     DIW 62;
      L     "MD100";
      SRW   3;
      L     2;
      +D;
      SLW   3;
      T     "MD100";
//;
      L     PID ["MD100"];	//; POSIZIONE ATTUALE
      T     #POSIZIONE_ATTUALE;
      L     "MD100";
      SRW   3;
      L     4;
      +D;
      SLW   3;
      T     "MD100";
//;
      L     PIW ["MD100"];	//;INGRESSI DIGITALI
      T     DIW 54;
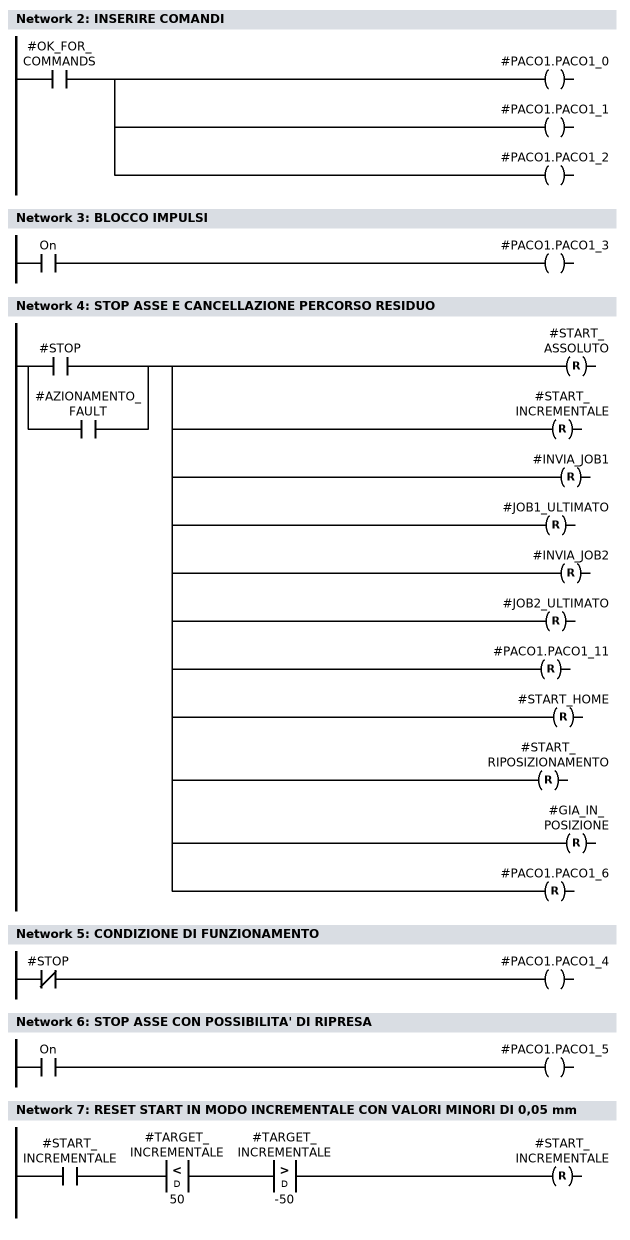
NETWORK
TITLE = INSERIRE COMANDI
      A     #OK_FOR_COMMANDS;
      =     #PACO1.PACO1_0;
      =     #PACO1.PACO1_1;
      =     #PACO1.PACO1_2;
NETWORK
TITLE = BLOCCO IMPULSI
      A     "On";
      =     #PACO1.PACO1_3;
NETWORK
TITLE = STOP ASSE E CANCELLAZIONE PERCORSO RESIDUO
      O     #STOP;
      O     #AZIONAMENTO_FAULT;
      R     #START_ASSOLUTO;
      R     #START_INCREMENTALE;
      R     #INVIA_JOB1;
      R     #JOB1_ULTIMATO;
      R     #INVIA_JOB2;
      R     #JOB2_ULTIMATO;
      R     #PACO1.PACO1_11;
      R     #START_HOME;
      R     #START_RIPOSIZIONAMENTO;
      R     #GIA_IN_POSIZIONE;
      R     #PACO1.PACO1_6;
NETWORK
TITLE = CONDIZIONE DI FUNZIONAMENTO
      AN    #STOP;
      =     #PACO1.PACO1_4;
NETWORK
TITLE = STOP ASSE CON POSSIBILITA' DI RIPRESA 
      A     "On";
      =     #PACO1.PACO1_5;
NETWORK
TITLE = RESET START IN MODO INCREMENTALE CON VALORI MINORI DI 0,05 mm
      A     #START_INCREMENTALE;
      A(;
      L     #TARGET_INCREMENTALE;
      L     50;
      <D;
      );
      A(;
      L     #TARGET_INCREMENTALE;
      L     -50;
      >D;
      );
      R     #START_INCREMENTALE;
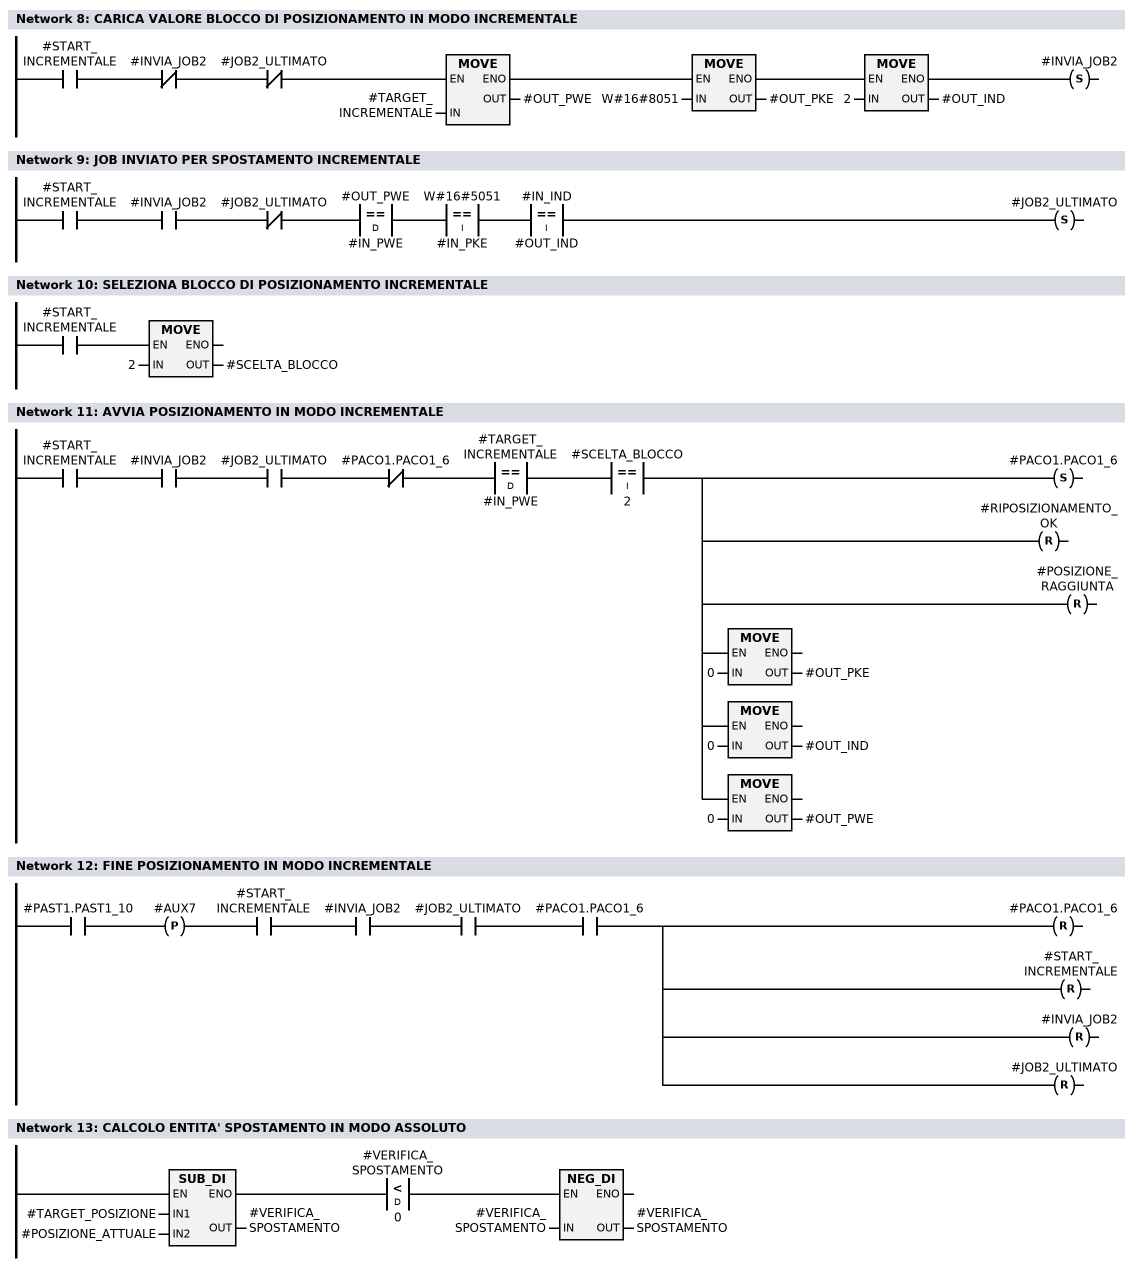
NETWORK
TITLE = CARICA VALORE BLOCCO DI POSIZIONAMENTO IN MODO INCREMENTALE
      A(;
      A(;
      A     #START_INCREMENTALE;
      AN    #INVIA_JOB2;
      AN    #JOB2_ULTIMATO;
      JNB   _001;
      L     #TARGET_INCREMENTALE;
      T     #OUT_PWE;
      SET;
      SAVE;
      CLR;
_001: A     BR;
      );
      JNB   _002;
      L     W#16#8051;
      T     #OUT_PKE;
      SET;
      SAVE;
      CLR;
_002: A     BR;
      );
      JNB   _003;
      L     2;
      T     #OUT_IND;
      SET;
      SAVE;
      CLR;
_003: A     BR;
      S     #INVIA_JOB2;
NETWORK
TITLE = JOB INVIATO PER SPOSTAMENTO INCREMENTALE
      A     #START_INCREMENTALE;
      A     #INVIA_JOB2;
      AN    #JOB2_ULTIMATO;
      A(;
      L     #OUT_PWE;
      L     #IN_PWE;
      ==D;
      );
      A(;
      L     W#16#5051;
      L     #IN_PKE;
      ==I;
      );
      A(;
      L     #IN_IND;
      L     #OUT_IND;
      ==I;
      );
      S     #JOB2_ULTIMATO;
NETWORK
TITLE = SELEZIONA BLOCCO DI POSIZIONAMENTO INCREMENTALE
      A     #START_INCREMENTALE;
      JNB   _004;
      L     2;
      T     #SCELTA_BLOCCO;
_004: NOP   0;
NETWORK
TITLE = AVVIA POSIZIONAMENTO IN MODO INCREMENTALE
      A     #START_INCREMENTALE;
      A     #INVIA_JOB2;
      A     #JOB2_ULTIMATO;
      AN    #PACO1.PACO1_6;
      A(;
      L     #TARGET_INCREMENTALE;
      L     #IN_PWE;
      ==D;
      );
      A(;
      L     #SCELTA_BLOCCO;
      L     2;
      ==I;
      );
      =     L 0.0;
      A     L 0.0;
      BLD   102;
      S     #PACO1.PACO1_6;
      A     L 0.0;
      BLD   102;
      R     #RIPOSIZIONAMENTO_OK;
      A     L 0.0;
      BLD   102;
      R     #POSIZIONE_RAGGIUNTA;
      A     L 0.0;
      JNB   _005;
      L     0;
      T     #OUT_PKE;
_005: NOP   0;
      A     L 0.0;
      JNB   _006;
      L     0;
      T     #OUT_IND;
_006: NOP   0;
      A     L 0.0;
      JNB   _007;
      L     0;
      T     #OUT_PWE;
_007: NOP   0;
NETWORK
TITLE = FINE POSIZIONAMENTO IN MODO INCREMENTALE
      A     #PAST1.PAST1_10;
      FP    #AUX7;
      A     #START_INCREMENTALE;
      A     #INVIA_JOB2;
      A     #JOB2_ULTIMATO;
      A     #PACO1.PACO1_6;
      R     #PACO1.PACO1_6;
      R     #START_INCREMENTALE;
      R     #INVIA_JOB2;
      R     #JOB2_ULTIMATO;
NETWORK
TITLE = CALCOLO ENTITA' SPOSTAMENTO IN MODO ASSOLUTO
      A(;
      L     #TARGET_POSIZIONE;
      L     #POSIZIONE_ATTUALE;
      -D;
      T     #VERIFICA_SPOSTAMENTO;
      AN    OV;
      SAVE;
      CLR;
      A     BR;
      );
      A(;
      L     #VERIFICA_SPOSTAMENTO;
      L     0;
      <D;
      );
      JNB   _008;
      L     #VERIFICA_SPOSTAMENTO;
      NEGD;
      T     #VERIFICA_SPOSTAMENTO;
_008: NOP   0;
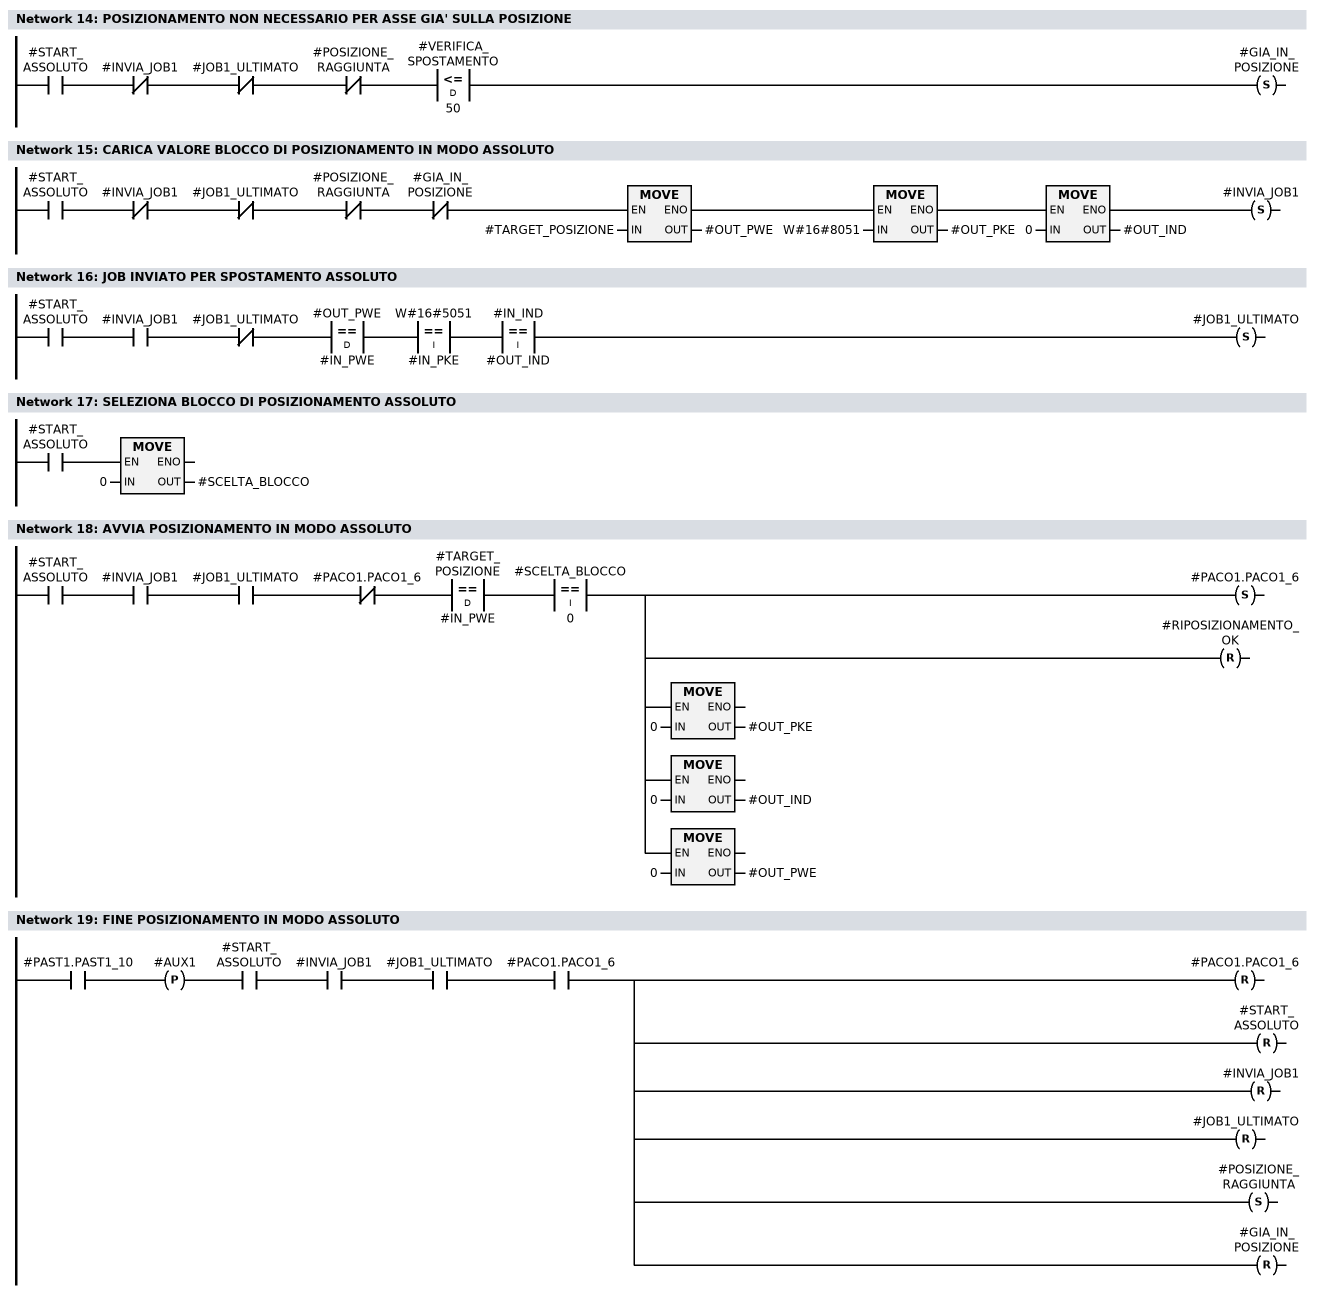
NETWORK
TITLE = POSIZIONAMENTO NON NECESSARIO PER ASSE GIA' SULLA POSIZIONE
      A     #START_ASSOLUTO;
      AN    #INVIA_JOB1;
      AN    #JOB1_ULTIMATO;
      AN    #POSIZIONE_RAGGIUNTA;
      A(;
      L     #VERIFICA_SPOSTAMENTO;
      L     50;
      <=D;
      );
      S     #GIA_IN_POSIZIONE;
NETWORK
TITLE = CARICA VALORE BLOCCO DI POSIZIONAMENTO IN MODO ASSOLUTO
      A(;
      A(;
      A     #START_ASSOLUTO;
      AN    #INVIA_JOB1;
      AN    #JOB1_ULTIMATO;
      AN    #POSIZIONE_RAGGIUNTA;
      AN    #GIA_IN_POSIZIONE;
      JNB   _009;
      L     #TARGET_POSIZIONE;
      T     #OUT_PWE;
      SET;
      SAVE;
      CLR;
_009: A     BR;
      );
      JNB   _00a;
      L     W#16#8051;
      T     #OUT_PKE;
      SET;
      SAVE;
      CLR;
_00a: A     BR;
      );
      JNB   _00b;
      L     0;
      T     #OUT_IND;
      SET;
      SAVE;
      CLR;
_00b: A     BR;
      S     #INVIA_JOB1;
NETWORK
TITLE = JOB INVIATO PER SPOSTAMENTO ASSOLUTO
      A     #START_ASSOLUTO;
      A     #INVIA_JOB1;
      AN    #JOB1_ULTIMATO;
      A(;
      L     #OUT_PWE;
      L     #IN_PWE;
      ==D;
      );
      A(;
      L     W#16#5051;
      L     #IN_PKE;
      ==I;
      );
      A(;
      L     #IN_IND;
      L     #OUT_IND;
      ==I;
      );
      S     #JOB1_ULTIMATO;
NETWORK
TITLE = SELEZIONA BLOCCO DI POSIZIONAMENTO ASSOLUTO
      A     #START_ASSOLUTO;
      JNB   _00c;
      L     0;
      T     #SCELTA_BLOCCO;
_00c: NOP   0;
NETWORK
TITLE = AVVIA POSIZIONAMENTO IN MODO ASSOLUTO
      A     #START_ASSOLUTO;
      A     #INVIA_JOB1;
      A     #JOB1_ULTIMATO;
      AN    #PACO1.PACO1_6;
      A(;
      L     #TARGET_POSIZIONE;
      L     #IN_PWE;
      ==D;
      );
      A(;
      L     #SCELTA_BLOCCO;
      L     0;
      ==I;
      );
      =     L 0.0;
      A     L 0.0;
      BLD   102;
      S     #PACO1.PACO1_6;
      A     L 0.0;
      BLD   102;
      R     #RIPOSIZIONAMENTO_OK;
      A     L 0.0;
      JNB   _00d;
      L     0;
      T     #OUT_PKE;
_00d: NOP   0;
      A     L 0.0;
      JNB   _00e;
      L     0;
      T     #OUT_IND;
_00e: NOP   0;
      A     L 0.0;
      JNB   _00f;
      L     0;
      T     #OUT_PWE;
_00f: NOP   0;
NETWORK
TITLE = FINE POSIZIONAMENTO IN MODO ASSOLUTO
      A     #PAST1.PAST1_10;
      FP    #AUX1;
      A     #START_ASSOLUTO;
      A     #INVIA_JOB1;
      A     #JOB1_ULTIMATO;
      A     #PACO1.PACO1_6;
      R     #PACO1.PACO1_6;
      R     #START_ASSOLUTO;
      R     #INVIA_JOB1;
      R     #JOB1_ULTIMATO;
      S     #POSIZIONE_RAGGIUNTA;
      R     #GIA_IN_POSIZIONE;
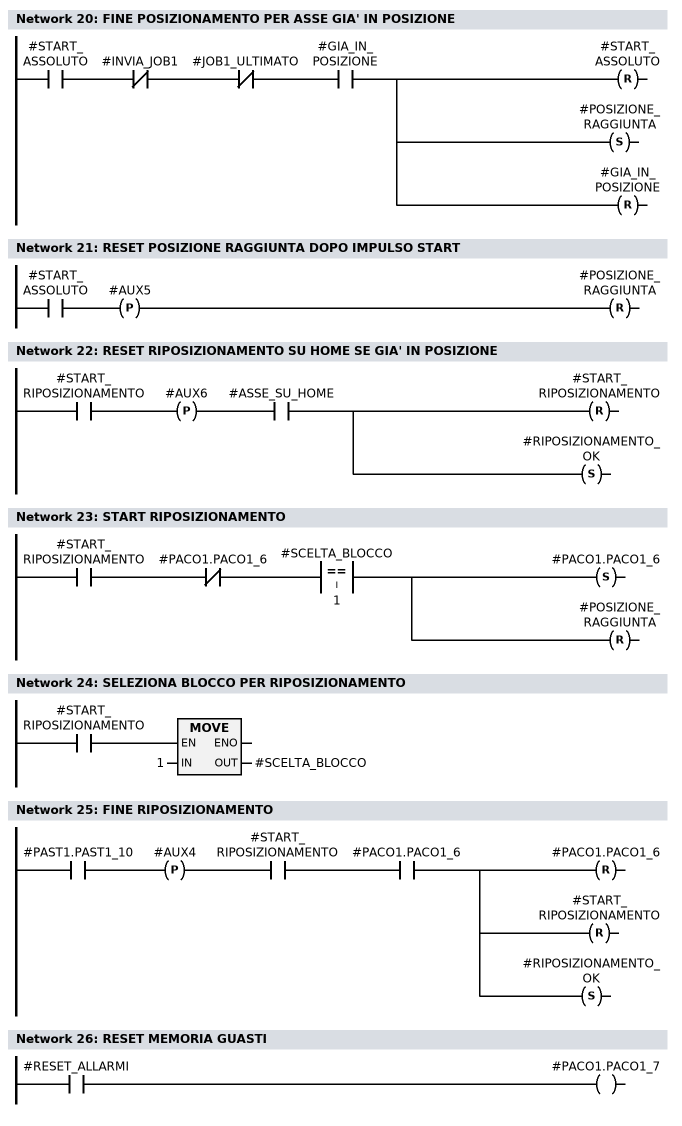
NETWORK
TITLE = FINE POSIZIONAMENTO PER ASSE GIA' IN POSIZIONE
      A     #START_ASSOLUTO;
      AN    #INVIA_JOB1;
      AN    #JOB1_ULTIMATO;
      A     #GIA_IN_POSIZIONE;
      R     #START_ASSOLUTO;
      S     #POSIZIONE_RAGGIUNTA;
      R     #GIA_IN_POSIZIONE;
NETWORK
TITLE = RESET POSIZIONE RAGGIUNTA DOPO IMPULSO START
      A     #START_ASSOLUTO;
      FP    #AUX5;
      R     #POSIZIONE_RAGGIUNTA;
NETWORK
TITLE = RESET RIPOSIZIONAMENTO SU HOME SE GIA' IN POSIZIONE
      A     #START_RIPOSIZIONAMENTO;
      FP    #AUX6;
      A     #ASSE_SU_HOME;
      R     #START_RIPOSIZIONAMENTO;
      S     #RIPOSIZIONAMENTO_OK;
NETWORK
TITLE = START RIPOSIZIONAMENTO
      A     #START_RIPOSIZIONAMENTO;
      AN    #PACO1.PACO1_6;
      A(;
      L     #SCELTA_BLOCCO;
      L     1;
      ==I;
      );
      S     #PACO1.PACO1_6;
      R     #POSIZIONE_RAGGIUNTA;
NETWORK
TITLE = SELEZIONA BLOCCO PER RIPOSIZIONAMENTO
      A     #START_RIPOSIZIONAMENTO;
      JNB   _010;
      L     1;
      T     #SCELTA_BLOCCO;
_010: NOP   0;
NETWORK
TITLE = FINE RIPOSIZIONAMENTO
      A     #PAST1.PAST1_10;
      FP    #AUX4;
      A     #START_RIPOSIZIONAMENTO;
      A     #PACO1.PACO1_6;
      R     #PACO1.PACO1_6;
      R     #START_RIPOSIZIONAMENTO;
      S     #RIPOSIZIONAMENTO_OK;
NETWORK
TITLE = RESET MEMORIA GUASTI
      A     #RESET_ALLARMI;
      =     #PACO1.PACO1_7;
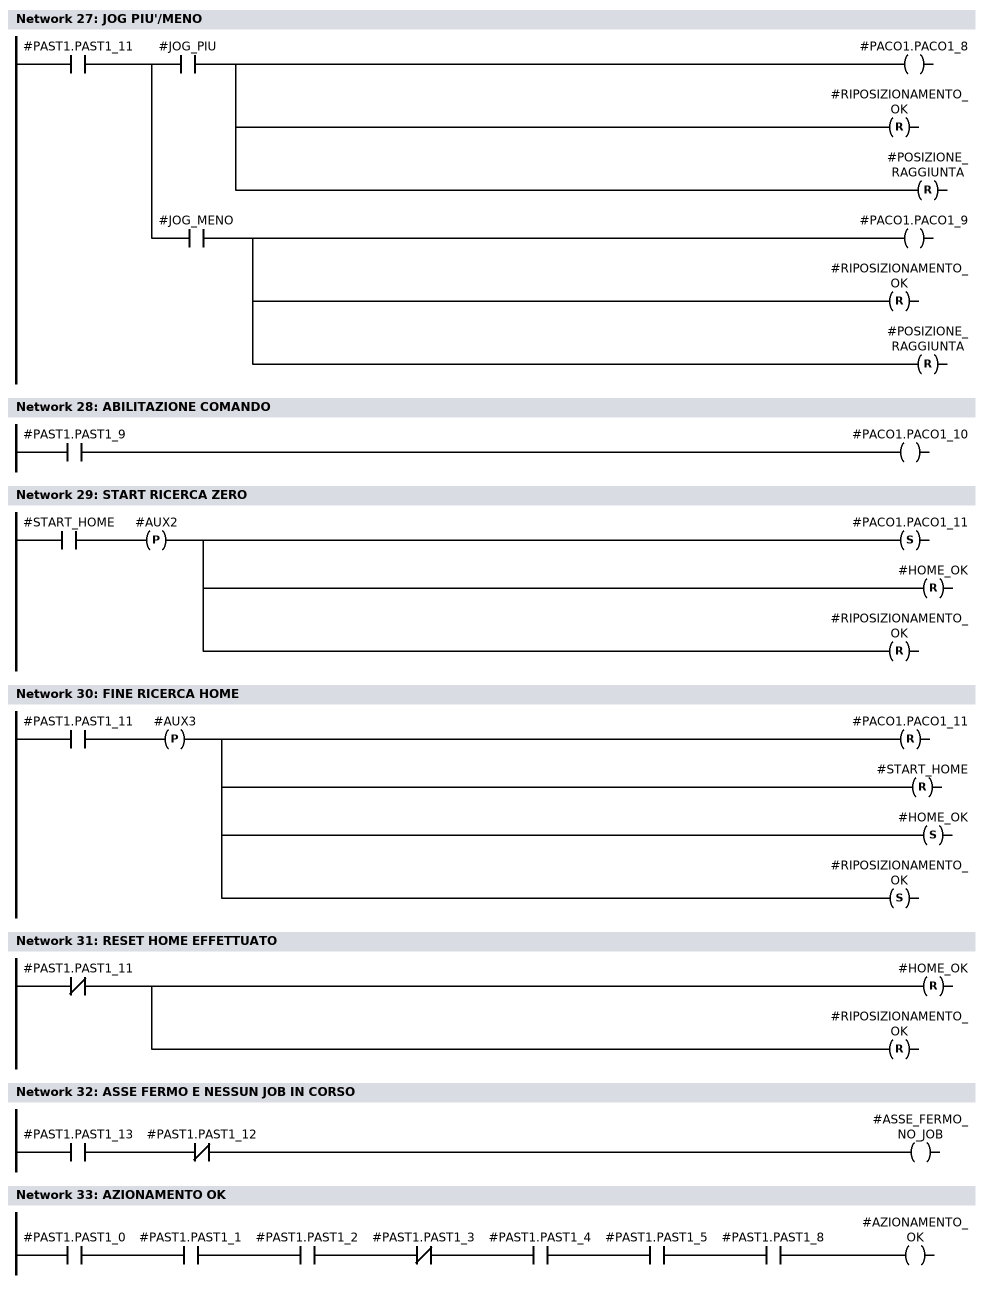
NETWORK
TITLE = JOG PIU'/MENO
      A     #PAST1.PAST1_11;
      =     L 1.0;
      A     L 1.0;
      A     #JOG_PIU;
      =     #PACO1.PACO1_8;
      R     #RIPOSIZIONAMENTO_OK;
      R     #POSIZIONE_RAGGIUNTA;
      A     L 1.0;
      A     #JOG_MENO;
      =     #PACO1.PACO1_9;
      R     #RIPOSIZIONAMENTO_OK;
      R     #POSIZIONE_RAGGIUNTA;
NETWORK
TITLE = ABILITAZIONE COMANDO
      A     #PAST1.PAST1_9;
      =     #PACO1.PACO1_10;
NETWORK
TITLE = START RICERCA ZERO
      A     #START_HOME;
      FP    #AUX2;
      S     #PACO1.PACO1_11;
      R     #HOME_OK;
      R     #RIPOSIZIONAMENTO_OK;
NETWORK
TITLE = FINE RICERCA HOME
      A     #PAST1.PAST1_11;
      FP    #AUX3;
      R     #PACO1.PACO1_11;
      R     #START_HOME;
      S     #HOME_OK;
      S     #RIPOSIZIONAMENTO_OK;
NETWORK
TITLE = RESET HOME EFFETTUATO
      AN    #PAST1.PAST1_11;
      R     #HOME_OK;
      R     #RIPOSIZIONAMENTO_OK;
NETWORK
TITLE = ASSE FERMO E NESSUN JOB IN CORSO
      A     #PAST1.PAST1_13;
      AN    #PAST1.PAST1_12;
      =     #ASSE_FERMO_NO_JOB;
NETWORK
TITLE = AZIONAMENTO OK
      A     #PAST1.PAST1_0;
      A     #PAST1.PAST1_1;
      A     #PAST1.PAST1_2;
      AN    #PAST1.PAST1_3;
      A     #PAST1.PAST1_4;
      A     #PAST1.PAST1_5;
      A     #PAST1.PAST1_8;
      =     #AZIONAMENTO_OK;
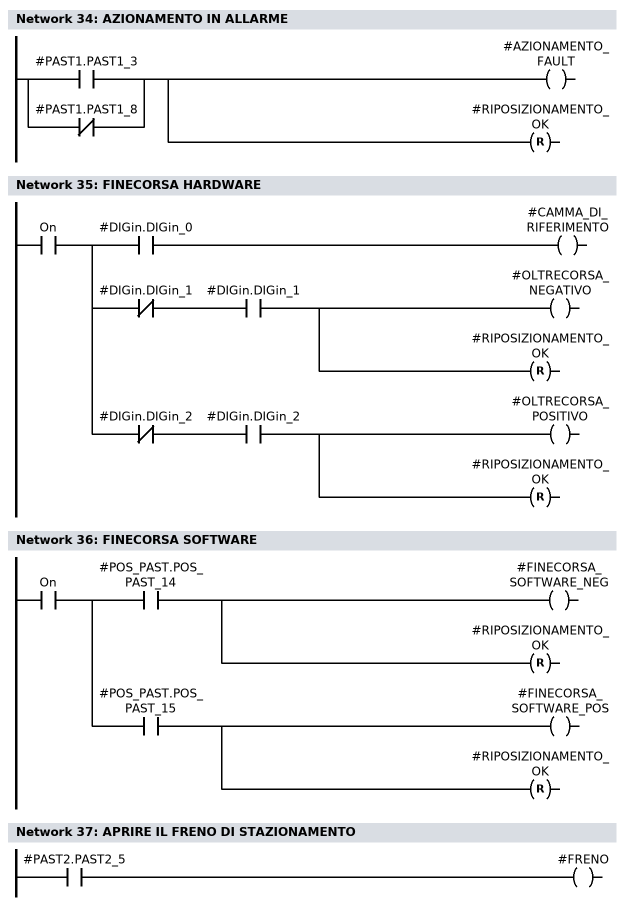
NETWORK
TITLE = AZIONAMENTO IN ALLARME
      O     #PAST1.PAST1_3;
      ON    #PAST1.PAST1_8;
      =     #AZIONAMENTO_FAULT;
      R     #RIPOSIZIONAMENTO_OK;
NETWORK
TITLE = FINECORSA HARDWARE
      A     "On";
      =     L 1.0;
      A     L 1.0;
      A     #DIGin.DIGin_0;
      =     #CAMMA_DI_RIFERIMENTO;
      A     L 1.0;
      AN    #DIGin.DIGin_1;
      A     #DIGin.DIGin_1;
      =     #OLTRECORSA_NEGATIVO;
      R     #RIPOSIZIONAMENTO_OK;
      A     L 1.0;
      AN    #DIGin.DIGin_2;
      A     #DIGin.DIGin_2;
      =     #OLTRECORSA_POSITIVO;
      R     #RIPOSIZIONAMENTO_OK;
NETWORK
TITLE = FINECORSA SOFTWARE
      A     "On";
      =     L 1.0;
      A     L 1.0;
      A     #POS_PAST.POS_PAST_14;
      =     #FINECORSA_SOFTWARE_NEG;
      R     #RIPOSIZIONAMENTO_OK;
      A     L 1.0;
      A     #POS_PAST.POS_PAST_15;
      =     #FINECORSA_SOFTWARE_POS;
      R     #RIPOSIZIONAMENTO_OK;
NETWORK
TITLE = APRIRE IL FRENO DI STAZIONAMENTO
      A     #PAST2.PAST2_5;
      =     #FRENO;
NETWORK
TITLE = AGGIORNAMENTO IMMAGINE USCITE
      L     #INDIRIZZO_INIZIALE_E_A;
      L     8;
      +I;
      SLD   3;
      T     "MD100";
      L     DIW 50;
      T     PQW ["MD100"];	//;PACO 1
      L     "MD100";
      SRW   3;
      L     2;
      +D;
      SLW   3;
      T     "MD100";
//;
      L     #SCELTA_BLOCCO;
      T     PQW ["MD100"];	//;SCELTA BLOCCO
      L     "MD100";
      SRW   3;
      L     6;
      +D;
      SLW   3;
      T     "MD100";
//;
      L     #OVERRIDE;
      T     PQW ["MD100"];	//;OVERRIDE
END_FUNCTION_BLOCK

// FC 7: know-how protected block, not included

FUNCTION "FC11 - STATUS" : VOID	// FC 11
TITLE = Sensors and proximity state
VERSION : 0.1
VAR_TEMP
  temp_INT : INT ;
END_VAR
BEGIN
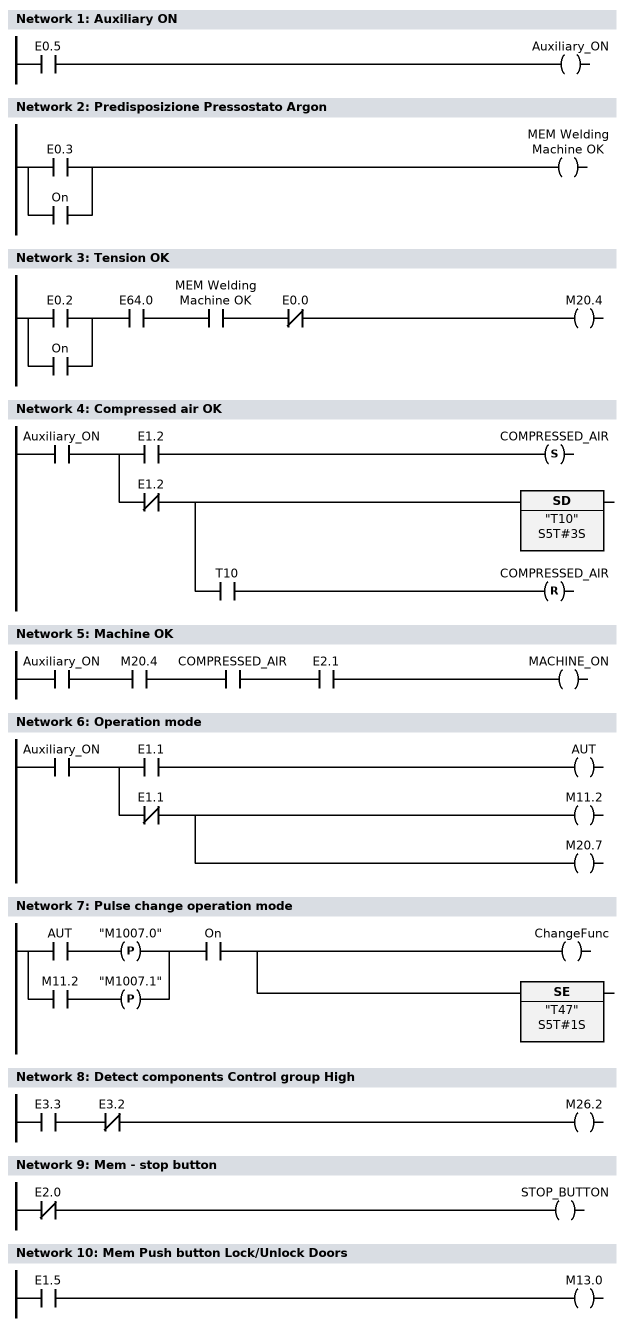
NETWORK
TITLE = Auxiliary ON
      A     "E0.5";
      =     "Auxiliary_ON";
NETWORK
TITLE = Predisposizione Pressostato Argon
      O     "E0.3";
      O     "On";
      =     "MEM Welding Machine OK";
NETWORK
TITLE = Tension OK
      A(;
      O     "E0.2";
      O     "On";
      );
      A     "E64.0";
      A     "MEM Welding Machine OK";
      AN    "E0.0";
      =     "M20.4";
NETWORK
TITLE = Compressed air OK
      A     "Auxiliary_ON";
      =     L 2.0;
      A     L 2.0;
      A     "E1.2";
      S     "COMPRESSED_AIR";
      A     L 2.0;
      AN    "E1.2";
      =     L 2.1;
      A     L 2.1;
      BLD   102;
      L     S5T#3S;
      SD    "T10";
      A     L 2.1;
      A     "T10";
      R     "COMPRESSED_AIR";
NETWORK
TITLE = Machine OK
      A     "Auxiliary_ON";
      A     "M20.4";
      A     "COMPRESSED_AIR";
      A     "E2.1";
      =     "MACHINE_ON";
NETWORK
TITLE = Operation mode
      A     "Auxiliary_ON";
      =     L 2.0;
      A     L 2.0;
      A     "E1.1";
      =     "AUT";
      A     L 2.0;
      AN    "E1.1";
      =     "M11.2";
      =     "M20.7";
NETWORK
TITLE = Pulse change operation mode
      A(;
      A     "AUT";
      FP    "M1007.0";
      O(;
      A     "M11.2";
      FP    "M1007.1";
      );
      );
      A     "On";
      =     "ChangeFunc";
      L     S5T#1S;
      SE    "T47";
NETWORK
TITLE = Detect components Control group High
      A     "E3.3";
      AN    "E3.2";
      =     "M26.2";
NETWORK
TITLE = Mem - stop button
      AN    "E2.0";
      =     "STOP_BUTTON";
NETWORK
TITLE = Mem Push button Lock/Unlock Doors
      A     "E1.5";
      =     "M13.0";
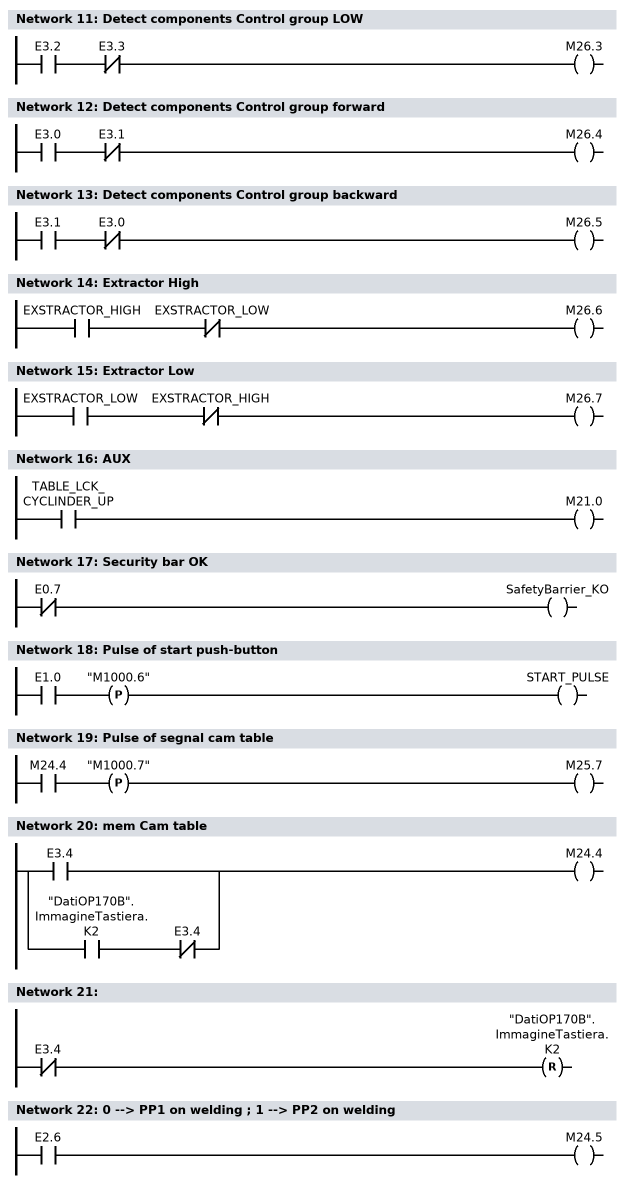
NETWORK
TITLE = Detect components Control group LOW
      A     "E3.2";
      AN    "E3.3";
      =     "M26.3";
NETWORK
TITLE = Detect components Control group forward
      A     "E3.0";
      AN    "E3.1";
      =     "M26.4";
NETWORK
TITLE = Detect components Control group backward
      A     "E3.1";
      AN    "E3.0";
      =     "M26.5";
NETWORK
TITLE = Extractor High
      A     "EXSTRACTOR_HIGH";
      AN    "EXSTRACTOR_LOW";
      =     "M26.6";
NETWORK
TITLE = Extractor Low
      A     "EXSTRACTOR_LOW";
      AN    "EXSTRACTOR_HIGH";
      =     "M26.7";
NETWORK
TITLE = AUX
      A     "TABLE_LCK_CYCLINDER_UP";
      =     "M21.0";
NETWORK
TITLE = Security bar OK
      AN    "E0.7";
      =     "SafetyBarrier_KO";
NETWORK
TITLE = Pulse of start push-button
      A     "E1.0";
      FP    "M1000.6";
      =     "START_PULSE";
NETWORK
TITLE = Pulse of segnal cam table
      A     "M24.4";
      FP    "M1000.7";
      =     "M25.7";
NETWORK
TITLE = mem Cam table
      O     "E3.4";
      O;
      A     "DatiOP170B".ImmagineTastiera.K2;
      AN    "E3.4";
      =     "M24.4";
NETWORK
TITLE =
      AN    "E3.4";
      R     "DatiOP170B".ImmagineTastiera.K2;
NETWORK
TITLE = 0 --> PP1 on welding ; 1 --> PP2 on welding
      A     "E2.6";
      =     "M24.5";
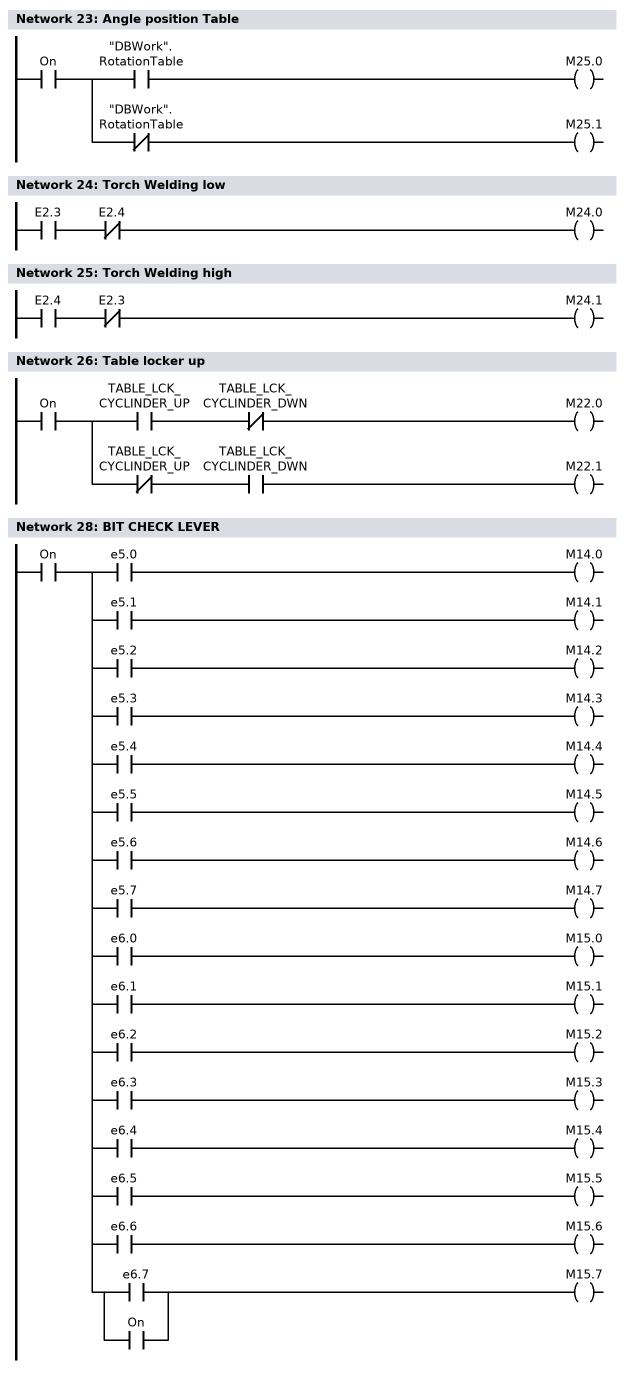
NETWORK
TITLE = Angle position Table
      A     "On";
      =     L 2.0;
      A     L 2.0;
      A     "DBWork".RotationTable;
      =     "M25.0";
      A     L 2.0;
      AN    "DBWork".RotationTable;
      =     "M25.1";
NETWORK
TITLE = Torch Welding low
      A     "E2.3";
      AN    "E2.4";
      =     "M24.0";
NETWORK
TITLE = Torch Welding high
      A     "E2.4";
      AN    "E2.3";
      =     "M24.1";
NETWORK
TITLE = Table locker up
      A     "On";
      =     L 2.0;
      A     L 2.0;
      A     "TABLE_LCK_CYCLINDER_UP";
      AN    "TABLE_LCK_CYCLINDER_DWN";
      =     "M22.0";
      A     L 2.0;
      AN    "TABLE_LCK_CYCLINDER_UP";
      A     "TABLE_LCK_CYCLINDER_DWN";
      =     "M22.1";
NETWORK
TITLE =
NETWORK
TITLE = BIT CHECK LEVER
      A     "On";
      =     L 2.0;
      A     L 2.0;
      A     "e5.0";
      =     "M14.0";
      A     L 2.0;
      A     "e5.1";
      =     "M14.1";
      A     L 2.0;
      A     "e5.2";
      =     "M14.2";
      A     L 2.0;
      A     "e5.3";
      =     "M14.3";
      A     L 2.0;
      A     "e5.4";
      =     "M14.4";
      A     L 2.0;
      A     "e5.5";
      =     "M14.5";
      A     L 2.0;
      A     "e5.6";
      =     "M14.6";
      A     L 2.0;
      A     "e5.7";
      =     "M14.7";
      A     L 2.0;
      A     "e6.0";
      =     "M15.0";
      A     L 2.0;
      A     "e6.1";
      =     "M15.1";
      A     L 2.0;
      A     "e6.2";
      =     "M15.2";
      A     L 2.0;
      A     "e6.3";
      =     "M15.3";
      A     L 2.0;
      A     "e6.4";
      =     "M15.4";
      A     L 2.0;
      A     "e6.5";
      =     "M15.5";
      A     L 2.0;
      A     "e6.6";
      =     "M15.6";
      A     L 2.0;
      A(;
      O     "e6.7";
      O     "On";
      );
      =     "M15.7";
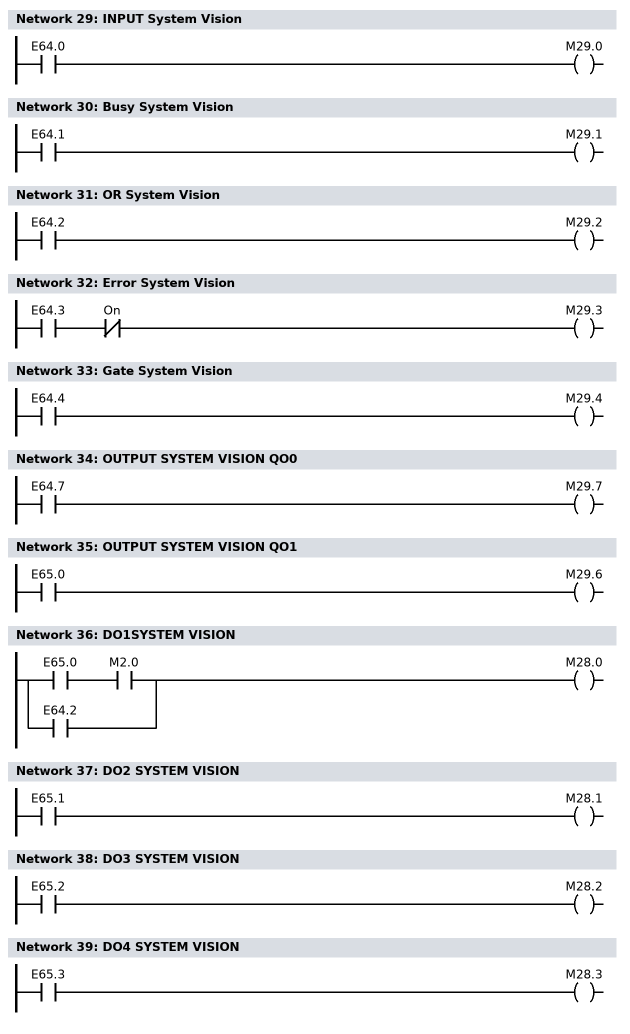
NETWORK
TITLE = INPUT System Vision 
      A     "E64.0";
      =     "M29.0";
NETWORK
TITLE = Busy System Vision
      A     "E64.1";
      =     "M29.1";
NETWORK
TITLE = OR System Vision
      A     "E64.2";
      =     "M29.2";
NETWORK
TITLE = Error System Vision
      A     "E64.3";
      AN    "On";
      =     "M29.3";
NETWORK
TITLE = Gate System Vision
      A     "E64.4";
      =     "M29.4";
NETWORK
TITLE = OUTPUT SYSTEM VISION QO0
      A     "E64.7";
      =     "M29.7";
NETWORK
TITLE = OUTPUT SYSTEM VISION QO1
      A     "E65.0";
      =     "M29.6";
NETWORK
TITLE = DO1SYSTEM VISION
      A     "E65.0";
      A     "M2.0";
      O     "E64.2";
      =     "M28.0";
NETWORK
TITLE = DO2 SYSTEM VISION
      A     "E65.1";
      =     "M28.1";
NETWORK
TITLE = DO3 SYSTEM VISION
      A     "E65.2";
      =     "M28.2";
NETWORK
TITLE = DO4 SYSTEM VISION
      A     "E65.3";
      =     "M28.3";
END_FUNCTION

FUNCTION "FC12 - GENERAL" : VOID	// FC 12
TITLE = General management
VERSION : 0.1
BEGIN
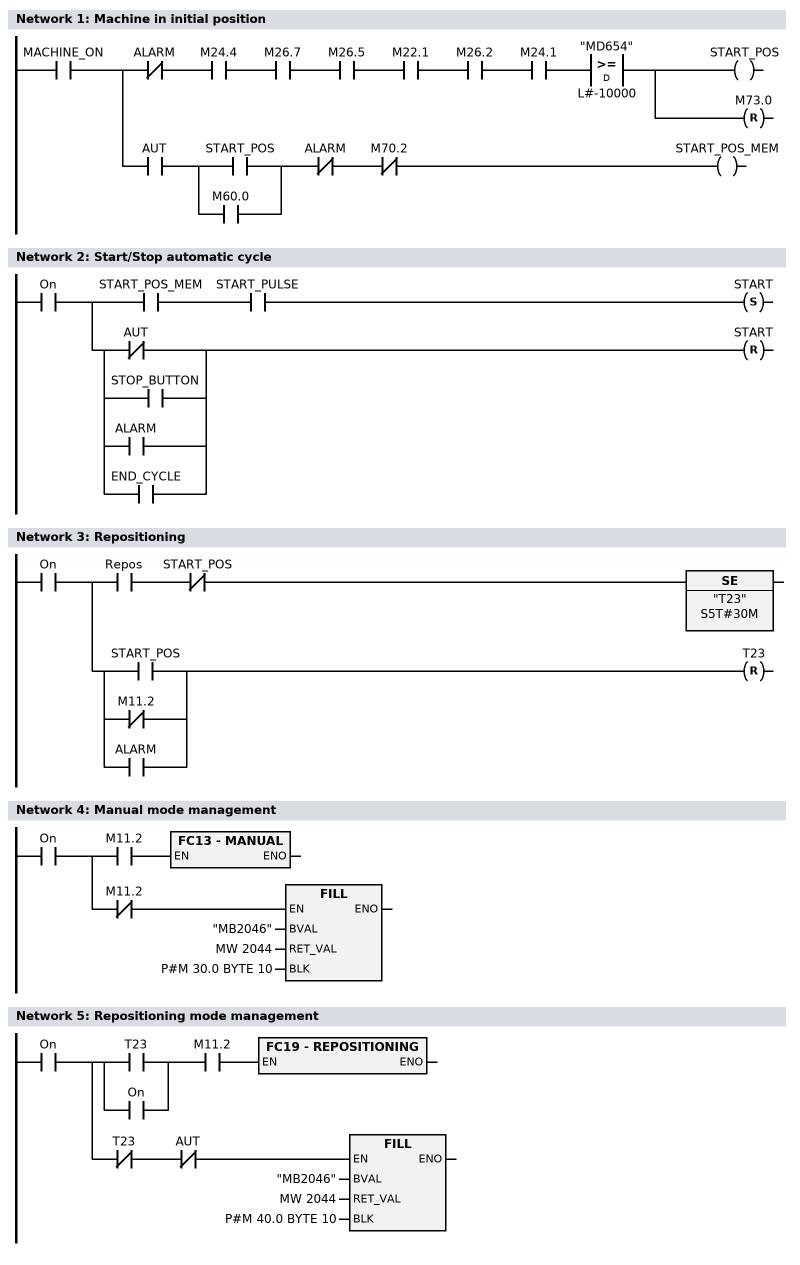
NETWORK
TITLE = Machine in initial position
      A     "MACHINE_ON";
      =     L 0.0;
      A     L 0.0;
      AN    "ALARM";
      A     "M24.4";
      A     "M26.7";
      A     "M26.5";
      A     "M22.1";
      A     "M26.2";
      A     "M24.1";
      A(;
      L     "MD654";
      L     L#-10000;
      >=D;
      );
      =     "START_POS";
      R     "M73.0";
      A     L 0.0;
      A     "AUT";
      A(;
      O     "START_POS";
      O     "M60.0";
      );
      AN    "ALARM";
      AN    "M70.2";
      =     "START_POS_MEM";
NETWORK
TITLE = Start/Stop automatic cycle
      A     "On";
      =     L 0.0;
      A     L 0.0;
      A     "START_POS_MEM";
      A     "START_PULSE";
      S     "START";
      A     L 0.0;
      A(;
      ON    "AUT";
      O     "STOP_BUTTON";
      O     "ALARM";
      O     "END_CYCLE";
      );
      R     "START";
NETWORK
TITLE = Repositioning
      A     "On";
      =     L 0.0;
      A     L 0.0;
      A     "Repos";
      AN    "START_POS";
      L     S5T#30M;
      SE    "T23";
      A     L 0.0;
      A(;
      O     "START_POS";
      ON    "M11.2";
      O     "ALARM";
      );
      R     "T23";
NETWORK
TITLE = Manual mode management
      A     "On";
      =     L 0.0;
      A     L 0.0;
      A     "M11.2";
      JNB   _001;
      CALL  "FC13 - MANUAL";
_001: NOP   0;
      A     L 0.0;
      AN    "M11.2";
      JNB   _002;
      CALL  "FILL" (
           BVAL                     := "MB2046",
           RET_VAL                  := MW 2044,
           BLK                      := P#M 30.0 BYTE 10);
_002: NOP   0;
NETWORK
TITLE = Repositioning mode management
      A     "On";
      =     L 0.0;
      A     L 0.0;
      A(;
      O     "T23";
      O     "On";
      );
      A     "M11.2";
      JNB   _003;
      CALL  "FC19 - REPOSITIONING";
_003: NOP   0;
      A     L 0.0;
      AN    "T23";
      AN    "AUT";
      JNB   _004;
      CALL  "FILL" (
           BVAL                     := "MB2046",
           RET_VAL                  := MW 2044,
           BLK                      := P#M 40.0 BYTE 10);
_004: NOP   0;
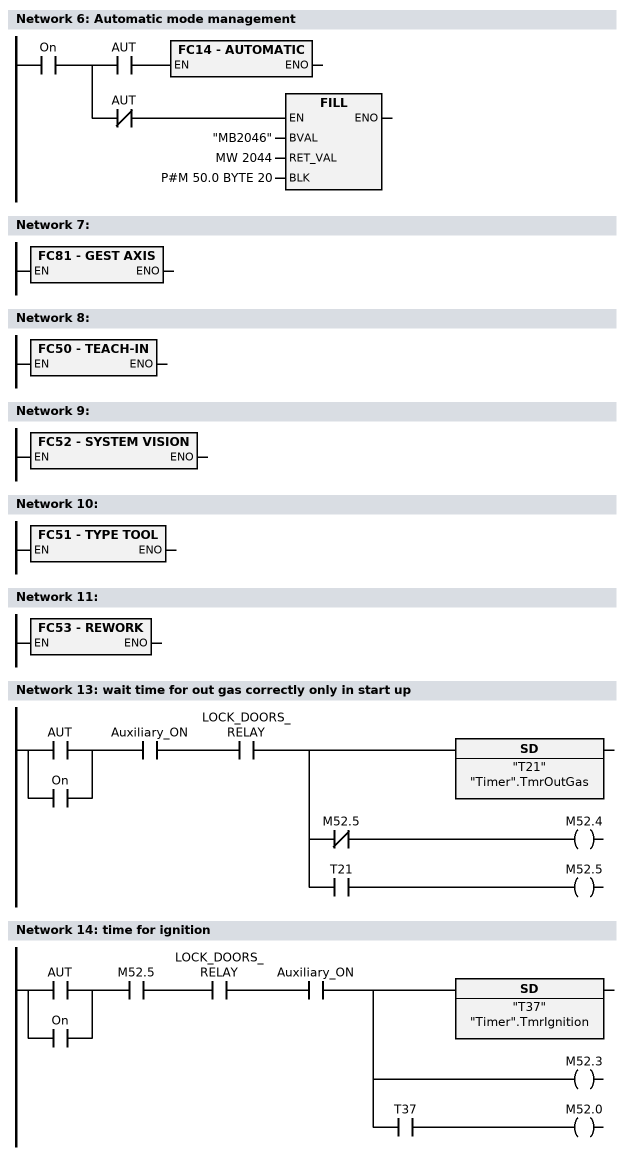
NETWORK
TITLE = Automatic mode management
//reset axis mouvement
      A     "On";
      =     L 0.0;
      A     L 0.0;
      A     "AUT";
      JNB   _005;
      CALL  "FC14 - AUTOMATIC";
_005: NOP   0;
      A     L 0.0;
      AN    "AUT";
      JNB   _006;
      CALL  "FILL" (
           BVAL                     := "MB2046",
           RET_VAL                  := MW 2044,
           BLK                      := P#M 50.0 BYTE 20);
_006: NOP   0;
NETWORK
TITLE =
      CALL  "FC81 - GEST AXIS";
      NOP   0;
NETWORK
TITLE =
      CALL  "FC50 - TEACH-IN";
      NOP   0;
NETWORK
TITLE =
      CALL  "FC52 - SYSTEM VISION";
      NOP   0;
NETWORK
TITLE =
//Controllo il tipo di portapezzo e carico i relativi dati
      CALL  "FC51 - TYPE TOOL";
      NOP   0;
NETWORK
TITLE =
      CALL  "FC53 - REWORK";
      NOP   0;
NETWORK
TITLE =
NETWORK
TITLE = wait time for out gas correctly only in start up 
//AUT - Tempo di attesa per avere gas in circolo e la torcia in temp
      A(;
      O     "AUT";
      O     "On";
      );
      A     "Auxiliary_ON";
      A     "LOCK_DOORS_RELAY";
      =     L 0.0;
      A     L 0.0;
      BLD   102;
      L     "Timer".TmrOutGas;
      SD    "T21";
      A     L 0.0;
      AN    "M52.5";
      =     "M52.4";
      A     L 0.0;
      A     "T21";
      =     "M52.5";
NETWORK
TITLE = time for ignition
      A(;
      O     "AUT";
      O     "On";
      );
      A     "M52.5";
      A     "LOCK_DOORS_RELAY";
      A     "Auxiliary_ON";
      =     L 0.0;
      A     L 0.0;
      BLD   102;
      L     "Timer".TmrIgnition;
      SD    "T37";
      A     L 0.0;
      BLD   102;
      =     "M52.3";
      A     L 0.0;
      A     "T37";
      =     "M52.0";
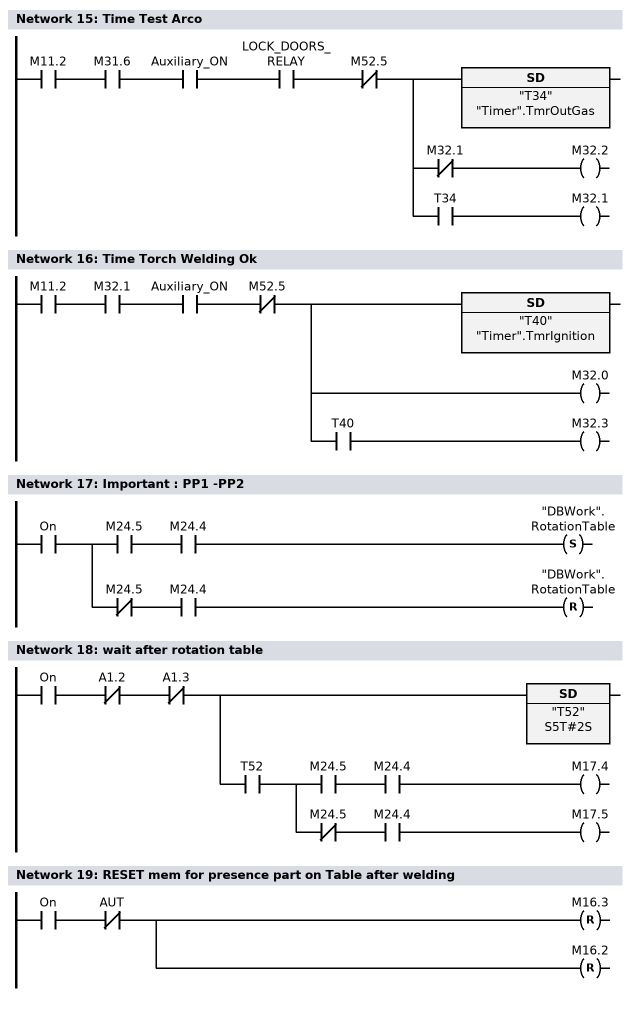
NETWORK
TITLE = Time Test Arco
//Test Arco Gas in Manuale
      A     "M11.2";
      A     "M31.6";
      A     "Auxiliary_ON";
      A     "LOCK_DOORS_RELAY";
      AN    "M52.5";
      =     L 0.0;
      A     L 0.0;
      BLD   102;
      L     "Timer".TmrOutGas;
      SD    "T34";
      A     L 0.0;
      AN    "M32.1";
      =     "M32.2";
      A     L 0.0;
      A     "T34";
      =     "M32.1";
NETWORK
TITLE = Time Torch Welding Ok
//Accensione Torcia in Manuale: per arrivare in Temp
      A     "M11.2";
      A     "M32.1";
      A     "Auxiliary_ON";
      AN    "M52.5";
      =     L 0.0;
      A     L 0.0;
      BLD   102;
      L     "Timer".TmrIgnition;
      SD    "T40";
      A     L 0.0;
      BLD   102;
      =     "M32.0";
      A     L 0.0;
      A     "T40";
      =     "M32.3";
NETWORK
TITLE = Important : PP1 -PP2 
      A     "On";
      =     L 0.0;
      A     L 0.0;
      A     "M24.5";
      A     "M24.4";
      S     "DBWork".RotationTable;
      A     L 0.0;
      AN    "M24.5";
      A     "M24.4";
      R     "DBWork".RotationTable;
NETWORK
TITLE = wait after rotation table
      A     "On";
      AN    "A1.2";
      AN    "A1.3";
      =     L 0.0;
      A     L 0.0;
      BLD   102;
      L     S5T#2S;
      SD    "T52";
      A     L 0.0;
      A     "T52";
      =     L 0.1;
      A     L 0.1;
      A     "M24.5";
      A     "M24.4";
      =     "M17.4";
      A     L 0.1;
      AN    "M24.5";
      A     "M24.4";
      =     "M17.5";
NETWORK
TITLE = RESET mem for presence part on Table after welding
      A     "On";
      AN    "AUT";
      R     "M16.3";
      R     "M16.2";
END_FUNCTION

